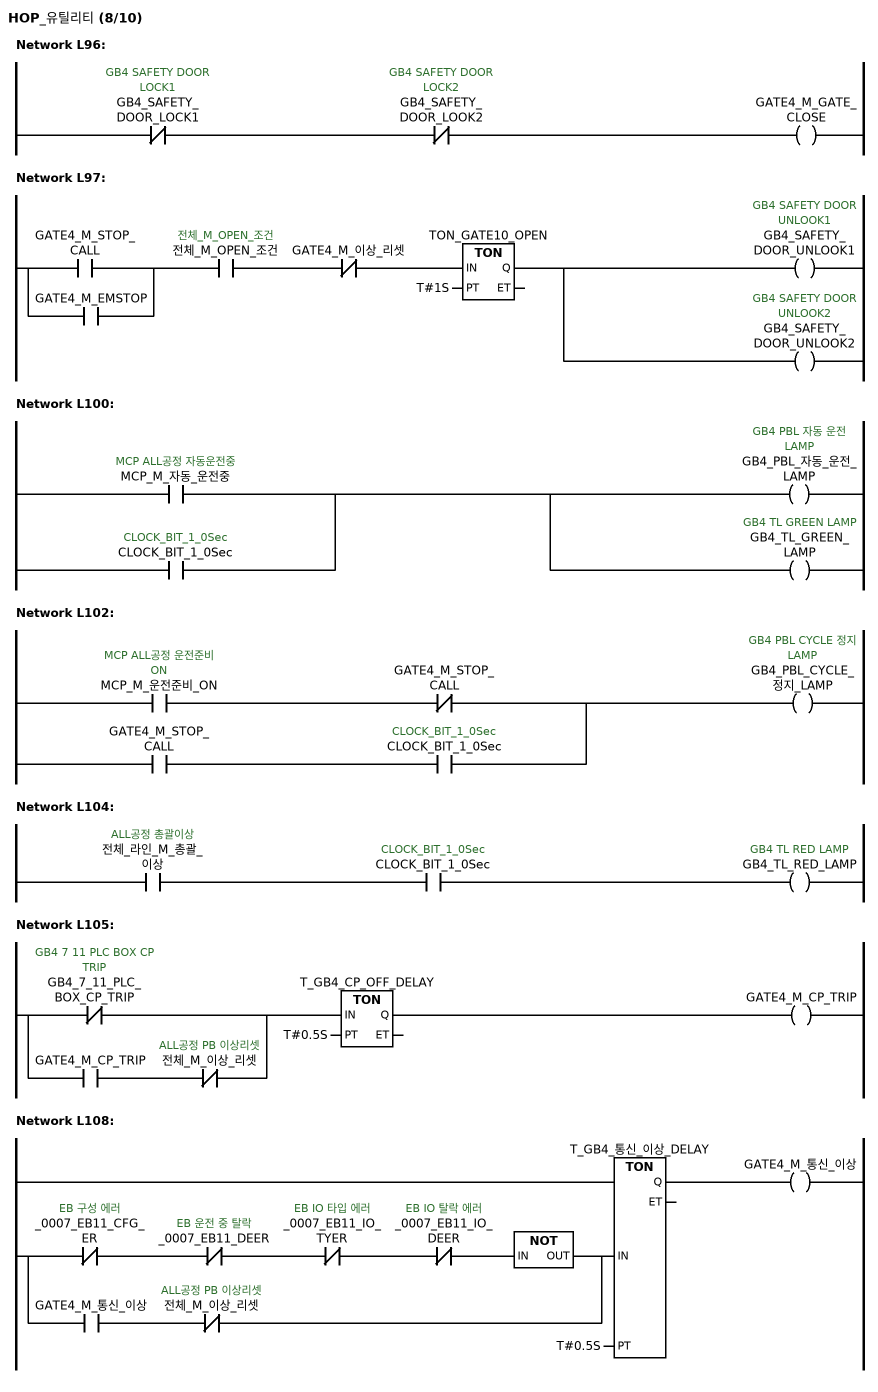
(* [picture p48: HOP_유틸리티 rungs L96-L108] *)
(* Rung L96 *)
GATE4_M_GATE_CLOSE := NOT GB4_SAFETY_DOOR_LOCK1 AND NOT GB4_SAFETY_DOOR_LOOK2;
(* Rung L97 *)
TON_GATE10_OPEN(IN := (GATE4_M_STOP_CALL OR GATE4_M_EMSTOP) AND 전체_M_OPEN_조건 AND NOT GATE4_M_이상_리셋, PT := T#1S);
GB4_SAFETY_DOOR_UNLOOK1 := TON_GATE10_OPEN.Q;
GB4_SAFETY_DOOR_UNLOOK2 := TON_GATE10_OPEN.Q;
(* Rung L100 *)
GB4_PBL_자동_운전_LAMP := MCP_M_자동_운전중 OR CLOCK_BIT_1_0Sec;
GB4_TL_GREEN_LAMP := MCP_M_자동_운전중 OR CLOCK_BIT_1_0Sec;
(* Rung L102 *)
GB4_PBL_CYCLE_정지_LAMP := (MCP_M_운전준비_ON AND NOT GATE4_M_STOP_CALL) OR (GATE4_M_STOP_CALL AND CLOCK_BIT_1_0Sec);
(* Rung L104 *)
GB4_TL_RED_LAMP := 전체_라인_M_총괄_이상 AND CLOCK_BIT_1_0Sec;
(* Rung L105 *)
T_GB4_CP_OFF_DELAY(IN := NOT GB4_7_11_PLC_BOX_CP_TRIP OR (GATE4_M_CP_TRIP AND NOT 전체_M_이상_리셋), PT := T#0.5S);
GATE4_M_CP_TRIP := T_GB4_CP_OFF_DELAY.Q;
(* Rung L108 *)
T_GB4_통신_이상_DELAY(IN := (NOT (NOT _0007_EB11_CFG_ER AND NOT _0007_EB11_DEER AND NOT _0007_EB11_IO_TYER AND NOT _0007_EB11_IO_DEER)) OR (GATE4_M_통신_이상 AND NOT 전체_M_이상_리셋), PT := T#0.5S);
GATE4_M_통신_이상 := T_GB4_통신_이상_DELAY.Q;

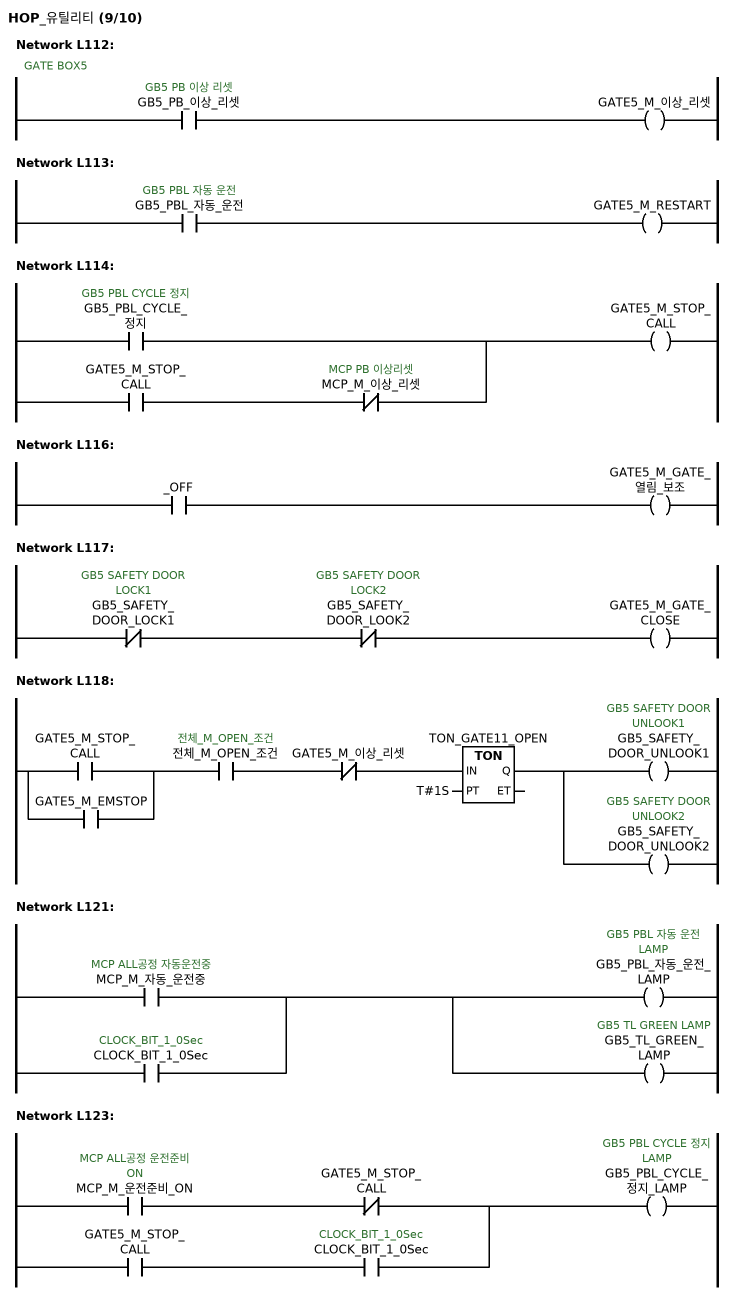
(* GATE BOX5 *)
(* Rung L112 *)
GATE5_M_이상_리셋 := GB5_PB_이상_리셋;
(* Rung L113 *)
GATE5_M_RESTART := GB5_PBL_자동_운전;
(* Rung L114 *)
GATE5_M_STOP_CALL := GB5_PBL_CYCLE_정지 OR (GATE5_M_STOP_CALL AND NOT MCP_M_이상_리셋);
(* Rung L116 *)
GATE5_M_GATE_열림_보조 := _OFF;
(* Rung L117 *)
GATE5_M_GATE_CLOSE := NOT GB5_SAFETY_DOOR_LOCK1 AND NOT GB5_SAFETY_DOOR_LOOK2;
(* Rung L118 *)
TON_GATE11_OPEN(IN := (GATE5_M_STOP_CALL OR GATE5_M_EMSTOP) AND 전체_M_OPEN_조건 AND NOT GATE5_M_이상_리셋, PT := T#1S);
GB5_SAFETY_DOOR_UNLOOK1 := TON_GATE11_OPEN.Q;
GB5_SAFETY_DOOR_UNLOOK2 := TON_GATE11_OPEN.Q;
(* Rung L121 *)
GB5_PBL_자동_운전_LAMP := MCP_M_자동_운전중 OR CLOCK_BIT_1_0Sec;
GB5_TL_GREEN_LAMP := MCP_M_자동_운전중 OR CLOCK_BIT_1_0Sec;
(* Rung L123 *)
GB5_PBL_CYCLE_정지_LAMP := (MCP_M_운전준비_ON AND NOT GATE5_M_STOP_CALL) OR (GATE5_M_STOP_CALL AND CLOCK_BIT_1_0Sec);

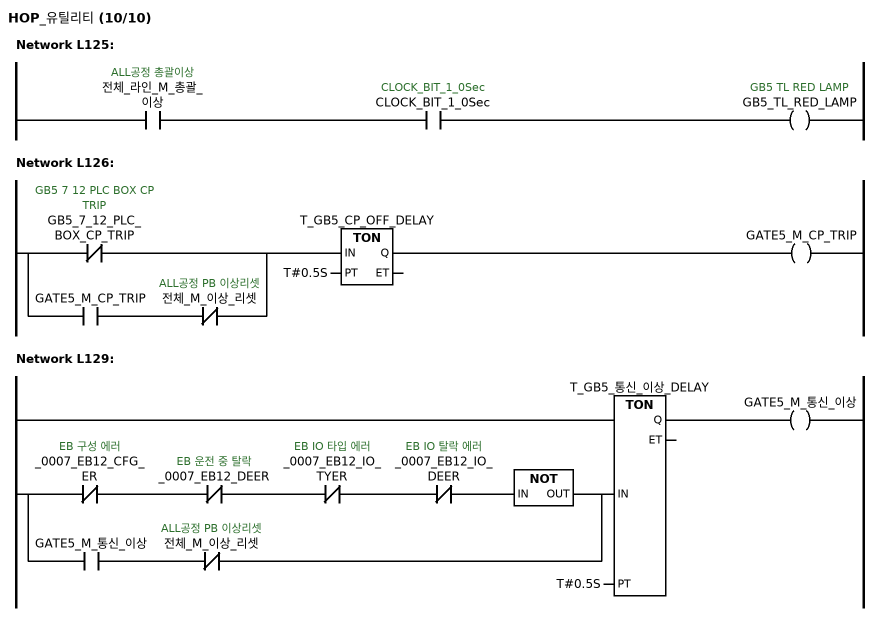
(* Rung L125 *)
GB5_TL_RED_LAMP := 전체_라인_M_총괄_이상 AND CLOCK_BIT_1_0Sec;
(* Rung L126 *)
T_GB5_CP_OFF_DELAY(IN := NOT GB5_7_12_PLC_BOX_CP_TRIP OR (GATE5_M_CP_TRIP AND NOT 전체_M_이상_리셋), PT := T#0.5S);
GATE5_M_CP_TRIP := T_GB5_CP_OFF_DELAY.Q;
(* Rung L129 *)
T_GB5_통신_이상_DELAY(IN := (NOT (NOT _0007_EB12_CFG_ER AND NOT _0007_EB12_DEER AND NOT _0007_EB12_IO_TYER AND NOT _0007_EB12_IO_DEER)) OR (GATE5_M_통신_이상 AND NOT 전체_M_이상_리셋), PT := T#0.5S);
GATE5_M_통신_이상 := T_GB5_통신_이상_DELAY.Q;
END_PROGRAM

PROGRAM 이상_총괄모음 (* task: 스캔 프로그램 *)
VAR_EXTERNAL RETAIN
    ALWAYS_OFF : BOOL; (* AT %MW3.0 *) (* 항시 OFF *)
    GATE1_M_CP_TRIP : BOOL; (* AT %MW400.15 *) (* GATEBOX1 CP OFF 이상 *)
    GATE1_M_EMSTOP : BOOL; (* AT %MW400.7 *) (* GATE1 비상정지 이상 *)
    GATE1_M_GATE_OPEN : BOOL; (* AT %MW400.13 *) (* GATEBOX1 이상 *)
    GATE1_M_통신_이상 : BOOL; (* AT %MW400.14 *) (* GATEBOX1 통신이상 *)
    GATE2_M_CP_TRIP : BOOL; (* AT %MW401.15 *) (* GATEBOX2 CP OFF 이상 *)
    GATE2_M_EMSTOP : BOOL; (* AT %MW401.7 *) (* GATE2 비상정지 이상 *)
    GATE2_M_GATE_OPEN : BOOL; (* AT %MW401.13 *) (* GATEBOX2 이상 *)
    GATE2_M_통신_이상 : BOOL; (* AT %MW401.14 *) (* GATEBOX2 통신이상 *)
    GATE3_M_CP_TRIP : BOOL; (* AT %MW402.15 *) (* GATEBOX3 CP OFF 이상 *)
    GATE3_M_EMSTOP : BOOL; (* AT %MW402.7 *) (* GATE3 비상정지 이상 *)
    GATE3_M_GATE_OPEN : BOOL; (* AT %MW402.13 *) (* GATEBOX3 이상 *)
    GATE3_M_통신_이상 : BOOL; (* AT %MW402.14 *) (* GATEBOX3 통신이상 *)
    GATE4_M_CP_TRIP : BOOL; (* AT %MW403.15 *)
    GATE4_M_EMSTOP : BOOL; (* AT %MW403.7 *)
    GATE4_M_GATE_OPEN : BOOL; (* AT %MW403.13 *)
    GATE4_M_통신_이상 : BOOL; (* AT %MW403.14 *)
    GATE5_M_CP_TRIP : BOOL; (* AT %MW404.15 *)
    GATE5_M_EMSTOP : BOOL; (* AT %MW404.7 *)
    GATE5_M_GATE_OPEN : BOOL; (* AT %MW404.13 *)
    GATE5_M_통신_이상 : BOOL; (* AT %MW404.14 *)
    HOP1_M_CP_OFF_이상 : BOOL; (* AT %MW360.15 *) (* HOP1 CP OFF 이상 *)
    HOP1_M_비상정지 : BOOL; (* AT %MW360.7 *) (* HOP1 비상정지 이상 *)
    HOP1_M_통신_이상 : BOOL; (* AT %MW360.14 *) (* HOP1 통신이상 *)
    INV1_M_CP_OFF_이상 : BOOL; (* AT %MW355.3 *) (* 인버터반1 CP OFF 이상 *)
    INV1_M_PS_DC_LOW : BOOL; (* AT %MW355.2 *) (* 인버터반1 PS저전압 이상 *)
    INV1_M_SPD_이상 : BOOL; (* AT %MW355.1 *) (* 인버터반1 SPD 이상 *)
    INV1_M_총괄_이상 : BOOL; (* AT %MW355.0 *) (* INV1_M_총괄_이상 *)
    INV1_M_통신_이상 : BOOL; (* AT %MW355.4 *) (* 인버터반1 통신이상 *)
    MCP_M_CP_OFF_이상 : BOOL; (* AT %MW351.0 *) (* MCP CP OFF 이상총괄 *)
    MCP_M_DISPLAY_CP_TRIP : BOOL; (* AT %MW351.6 *) (* MCP 출력전원 CP OFF 이상 *)
    MCP_M_HUB_CP_TRIP : BOOL; (* AT %MW351.1 *) (* MCP PS전원 CP OFF 이상 *)
    MCP_M_INPUT_CP_TRIP : BOOL; (* AT %MW351.3 *) (* MCP HUB전원  CP OFF 이상 *)
    MCP_M_OUTPUT_CP_TRIP : BOOL; (* AT %MW351.4 *) (* MCP 통신모듈 전원 CP OFF 이상 *)
    MCP_M_OUTPUT_MC_이상 : BOOL; (* AT %MW354.8 *) (* MCP 운전준비 MC 이상 *)
    MCP_M_PROFI_PWR_CP_TRIP : BOOL; (* AT %MW351.5 *) (* MCP 입력전원 CP OFF 이상 *)
    MCP_M_PS1_DC_LOW : BOOL; (* AT %MW353.1 *) (* MCP PS1 전원 이상 *)
    MCP_M_PS2_DC_LOW : BOOL; (* AT %MW353.2 *) (* MCP PS2 전원 이상 *)
    MCP_M_PS3_DC_LOW : BOOL; (* AT %MW353.3 *) (* MCP PS3 전원 이상 *)
    MCP_M_PS4_DC_LOW : BOOL; (* AT %MW353.4 *) (* MCP PS4 전원 이상 *)
    MCP_M_PS_DC_LOW : BOOL; (* AT %MW353.0 *) (* MCP PS 전원 이상총괄 *)
    MCP_M_SAG1_1_이상 : BOOL; (* AT %MW352.1 *) (* MCP SAG장치 이상 *)
    MCP_M_SAG1_2_이상 : BOOL; (* AT %MW352.2 *) (* MC SAG장치2 이상 *)
    MCP_M_SAG_이상 : BOOL; (* AT %MW352.0 *) (* MCP SAG장치 이상총괄 *)
    MCP_M_SPD_이상 : BOOL; (* AT %MW354.0 *) (* MCP 동력반 SPD 이상 *)
    MCP_M_비상정지 : BOOL; (* AT %MW350.7 *) (* MCP 비상정지 이상 *)
    MCP_M_이상_리셋 : BOOL; (* AT %MW350.4 *) (* MCP PB 이상리셋 *)
    MCP_M_통신_CP_TRIP : BOOL; (* AT %MW351.2 *) (* MCP   HMI전원  CP OFF 이상 *)
    MCP_M_통신_이상 : BOOL; (* AT %MW352.8 *) (* MCP 통신이상 *)
    S362_M_총괄_CP_이상 : BOOL; (* AT %MW1009.7 *) (* S362 CP OFF 이상 *)
    S362_M_총괄_CT_이상 : BOOL; (* AT %MW1010.4 *) (* S362   TACK TIME 이상 *)
    S362_M_총괄_INV_이상 : BOOL; (* AT %MW1009.9 *) (* S362 인버터 이상 *)
    S362_M_총괄_LS_이상 : BOOL; (* AT %MW1009.15 *) (* S362 LS 이상 *)
    S362_M_총괄_MATCH_이상 : BOOL; (* AT %MW1010.0 *) (* S362 매트SW 이상 *)
    S362_M_총괄_MC_이상 : BOOL; (* AT %MW1009.13 *) (* S362 MC 이상 *)
    S362_M_총괄_MOTOR_이상 : BOOL; (* AT %MW1010.3 *) (* S362 MOTOR 이상 *)
    S362_M_총괄_NFB_이상 : BOOL; (* AT %MW1009.11 *) (* S362 NFB 이상 *)
    S362_M_총괄_ROBOT_이상 : BOOL; (* AT %MW1010.1 *) (* S362 ROBOT 이상 *)
    S362_M_총괄_SAFETY_이상 : BOOL; (* AT %MW1009.2 *) (* S362 SAFETY 이상 *)
    S362_M_총괄_공기압_이상 : BOOL; (* AT %MW1009.3 *) (* S362 공기압 이상 *)
    S362_M_총괄_비상정지_이상 : BOOL; (* AT %MW1009.1 *) (* S362_M_총괄_비상정지_이상 *)
    S362_M_총괄_사양_이상 : BOOL; (* AT %MW1009.6 *) (* S362 사양 이상 *)
    S362_M_총괄_오버런_이상 : BOOL; (* AT %MW1009.12 *) (* S362 OVER RUN 이상 *)
    S362_M_총괄_용접타점수_이상 : BOOL; (* AT %MW1010.2 *) (* S362 용접타점수 이상 *)
    S362_M_총괄_제품감지_이상 : BOOL; (* AT %MW1009.4 *) (* S362 제품감지 이상 *)
    S362_M_총괄_차종_이상 : BOOL; (* AT %MW1009.5 *) (* S362 차종 이상 *)
    S362_M_총괄_통신_이상 : BOOL; (* AT %MW1009.14 *) (* S362 통신이상 *)
    S364_M_총괄_CP_이상 : BOOL; (* AT %MW2009.7 *) (* S364 CP OFF 이상 *)
    S364_M_총괄_CT_이상 : BOOL; (* AT %MW2010.4 *) (* S364   TACK TIME 이상 *)
    S364_M_총괄_LS_이상 : BOOL; (* AT %MW2009.15 *) (* S364 LS 이상 *)
    S364_M_총괄_MATCH_이상 : BOOL; (* AT %MW2010.0 *) (* S364 매트SW 이상 *)
    S364_M_총괄_ROBOT_이상 : BOOL; (* AT %MW2010.1 *) (* S364 ROBOT 이상 *)
    S364_M_총괄_SAFETY_이상 : BOOL; (* AT %MW2009.2 *) (* S364 SAFETY 이상 *)
    S364_M_총괄_공기압_이상 : BOOL; (* AT %MW2009.3 *) (* S364 공기압 이상 *)
    S364_M_총괄_비상정지_이상 : BOOL; (* AT %MW2009.1 *) (* S364_M_총괄_비상정지_이상 *)
    S364_M_총괄_사양_이상 : BOOL; (* AT %MW2009.6 *) (* S364 사양 이상 *)
    S364_M_총괄_용접타점수_이상 : BOOL; (* AT %MW2010.2 *) (* S364 용접타점수 이상 *)
    S364_M_총괄_제품감지_이상 : BOOL; (* AT %MW2009.4 *) (* S364 제품감지 이상 *)
    S364_M_총괄_차종_이상 : BOOL; (* AT %MW2009.5 *) (* S364 차종 이상 *)
    S364_M_총괄_통신_이상 : BOOL; (* AT %MW2009.14 *) (* S364 통신이상 *)
    S365_M_총괄_CP_이상 : BOOL; (* AT %MW2509.7 *) (* S365 CP OFF 이상 *)
    S365_M_총괄_CT_이상 : BOOL; (* AT %MW2510.4 *) (* S365   TACK TIME 이상 *)
    S365_M_총괄_LS_이상 : BOOL; (* AT %MW2509.15 *) (* S365 LS 이상 *)
    S365_M_총괄_MATCH_이상 : BOOL; (* AT %MW2510.0 *) (* S365 매트SW 이상 *)
    S365_M_총괄_ROBOT_이상 : BOOL; (* AT %MW2510.1 *) (* S365 ROBOT 이상 *)
    S365_M_총괄_SAFETY_이상 : BOOL; (* AT %MW2509.2 *) (* S365 SAFETY 이상 *)
    S365_M_총괄_공기압_이상 : BOOL; (* AT %MW2509.3 *) (* S365 공기압 이상 *)
    S365_M_총괄_비상정지_이상 : BOOL; (* AT %MW2509.1 *) (* S365_M_총괄_비상정지_이상 *)
    S365_M_총괄_사양_이상 : BOOL; (* AT %MW2509.6 *) (* S365 사양 이상 *)
    S365_M_총괄_용접타점수_이상 : BOOL; (* AT %MW2510.2 *) (* S365 용접타점수 이상 *)
    S365_M_총괄_제품감지_이상 : BOOL; (* AT %MW2509.4 *) (* S365 제품감지 이상 *)
    S365_M_총괄_차종_이상 : BOOL; (* AT %MW2509.5 *) (* S365 차종 이상 *)
    S365_M_총괄_통신_이상 : BOOL; (* AT %MW2509.14 *) (* S365 통신이상 *)
    S366_M_총괄_CP_이상 : BOOL; (* AT %MW3009.7 *) (* S366 CP OFF 이상 *)
    S366_M_총괄_CT_이상 : BOOL; (* AT %MW3010.4 *) (* S366   TACK TIME 이상 *)
    S366_M_총괄_INV_이상 : BOOL; (* AT %MW3009.9 *) (* S366 인버터 이상 *)
    S366_M_총괄_LS_이상 : BOOL; (* AT %MW3009.15 *) (* S366 LS 이상 *)
    S366_M_총괄_MATCH_이상 : BOOL; (* AT %MW3010.0 *) (* S366 매트SW 이상 *)
    S366_M_총괄_MC_이상 : BOOL; (* AT %MW3009.13 *) (* S366 MC 이상 *)
    S366_M_총괄_MOTOR_이상 : BOOL; (* AT %MW3010.3 *) (* S366 MOTOR 이상 *)
    S366_M_총괄_NFB_이상 : BOOL; (* AT %MW3009.11 *) (* S366 NFB 이상 *)
    S366_M_총괄_ROBOT_이상 : BOOL; (* AT %MW3010.1 *) (* S366 ROBOT 이상 *)
    S366_M_총괄_SAFETY_이상 : BOOL; (* AT %MW3009.2 *) (* S366_M_총괄_SAFETY_이상 *)
    S366_M_총괄_공기압_이상 : BOOL; (* AT %MW3009.3 *) (* S366 공기압 이상 *)
    S366_M_총괄_비상정지_이상 : BOOL; (* AT %MW3009.1 *) (* S366_M_총괄_비상정지_이상 *)
    S366_M_총괄_사양_이상 : BOOL; (* AT %MW3009.6 *) (* S366 사양 이상 *)
    S366_M_총괄_오버런_이상 : BOOL; (* AT %MW3009.12 *) (* S366 OVER RUN 이상 *)
    S366_M_총괄_용접타점수_이상 : BOOL; (* AT %MW3010.2 *) (* S366 용접타점수 이상 *)
    S366_M_총괄_제품감지_이상 : BOOL; (* AT %MW3009.4 *) (* S366 제품감지 이상 *)
    S366_M_총괄_차종_이상 : BOOL; (* AT %MW3009.5 *) (* S366 차종 이상 *)
    S366_M_총괄_통신_이상 : BOOL; (* AT %MW3009.14 *) (* S366 통신이상 *)
    S367_M_총괄_CP_이상 : BOOL; (* AT %MW3509.7 *) (* S367 CP OFF 이상 *)
    S367_M_총괄_CT_이상 : BOOL; (* AT %MW3510.4 *) (* S367   TACK TIME 이상 *)
    S367_M_총괄_LS_이상 : BOOL; (* AT %MW3509.15 *) (* S367 LS 이상 *)
    S367_M_총괄_MATCH_이상 : BOOL; (* AT %MW3510.0 *) (* S367 매트SW 이상 *)
    S367_M_총괄_ROBOT_이상 : BOOL; (* AT %MW3510.1 *) (* S367 ROBOT 이상 *)
    S367_M_총괄_SAFETY_이상 : BOOL; (* AT %MW3509.2 *) (* S367_M_총괄_SAFETY_이상 *)
    S367_M_총괄_공기압_이상 : BOOL; (* AT %MW3509.3 *) (* S367 공기압 이상 *)
    S367_M_총괄_비상정지_이상 : BOOL; (* AT %MW3509.1 *) (* S367_M_총괄_비상정지_이상 *)
    S367_M_총괄_사양_이상 : BOOL; (* AT %MW3509.6 *) (* S367 사양 이상 *)
    S367_M_총괄_용접타점수_이상 : BOOL; (* AT %MW3510.2 *) (* S367 용접타점수 이상 *)
    S367_M_총괄_제품감지_이상 : BOOL; (* AT %MW3509.4 *) (* S367 제품감지 이상 *)
    S367_M_총괄_차종_이상 : BOOL; (* AT %MW3509.5 *) (* S367 차종 이상 *)
    S367_M_총괄_통신_이상 : BOOL; (* AT %MW3509.14 *) (* S367 통신이상 *)
    S368_M_총괄_CP_이상 : BOOL; (* AT %MW4009.7 *) (* S368 CP OFF 이상 *)
    S368_M_총괄_CT_이상 : BOOL; (* AT %MW4010.4 *) (* S368   TACK TIME 이상 *)
    S368_M_총괄_LS_이상 : BOOL; (* AT %MW4009.15 *) (* S368 LS 이상 *)
    S368_M_총괄_MATCH_이상 : BOOL; (* AT %MW4010.0 *) (* S368 매트SW 이상 *)
    S368_M_총괄_ROBOT_이상 : BOOL; (* AT %MW4010.1 *) (* S368 ROBOT 이상 *)
    S368_M_총괄_SAFETY_이상 : BOOL; (* AT %MW4009.2 *) (* S368_M_총괄_SAFETY_이상 *)
    S368_M_총괄_공기압_이상 : BOOL; (* AT %MW4009.3 *) (* S368 공기압 이상 *)
    S368_M_총괄_비상정지_이상 : BOOL; (* AT %MW4009.1 *) (* S368_M_총괄_비상정지_이상 *)
    S368_M_총괄_사양_이상 : BOOL; (* AT %MW4009.6 *) (* S368 사양 이상 *)
    S368_M_총괄_용접타점수_이상 : BOOL; (* AT %MW4010.2 *) (* S368 용접타점수 이상 *)
    S368_M_총괄_제품감지_이상 : BOOL; (* AT %MW4009.4 *) (* S368 제품감지 이상 *)
    S368_M_총괄_차종_이상 : BOOL; (* AT %MW4009.5 *) (* S368 차종 이상 *)
    S368_M_총괄_통신_이상 : BOOL; (* AT %MW4009.14 *) (* S368 통신이상 *)
    S369_1_M_총괄_CP_이상 : BOOL; (* AT %MW4509.7 *) (* S369-1 CP OFF 이상 *)
    S369_1_M_총괄_CT_이상 : BOOL; (* AT %MW4510.4 *) (* S369-1 TACK TIME 이상 *)
    S369_1_M_총괄_LS_이상 : BOOL; (* AT %MW4509.15 *) (* S369-1 LS 이상 *)
    S369_1_M_총괄_MATCH_이상 : BOOL; (* AT %MW4510.0 *) (* S369-1 매트SW 이상 *)
    S369_1_M_총괄_ROBOT_이상 : BOOL; (* AT %MW4510.1 *) (* S369-1 ROBOT 이상 *)
    S369_1_M_총괄_SAFETY_이상 : BOOL; (* AT %MW4509.2 *) (* S369_1_M_총괄_SAFETY_이상 *)
    S369_1_M_총괄_공기압_이상 : BOOL; (* AT %MW4509.3 *) (* S36-1 공기압 이상 *)
    S369_1_M_총괄_사양_이상 : BOOL; (* AT %MW4509.6 *) (* S369-1 사양 이상 *)
    S369_1_M_총괄_용접타점수_이상 : BOOL; (* AT %MW4510.2 *) (* S369-1 용접타점수 이상 *)
    S369_1_M_총괄_제품감지_이상 : BOOL; (* AT %MW4509.4 *) (* S369-1 제품감지 이상 *)
    S369_1_M_총괄_차종_이상 : BOOL; (* AT %MW4509.5 *) (* S369-1 차종 이상 *)
    S369_1_M_총괄_통신_이상 : BOOL; (* AT %MW4509.14 *) (* S369-1 통신이상 *)
    S369_M_총괄_CP_이상 : BOOL; (* AT %MW5009.7 *) (* S369 CP OFF 이상 *)
    S369_M_총괄_CT_이상 : BOOL; (* AT %MW5010.4 *) (* S369   TACK TIME 이상 *)
    S369_M_총괄_LS_이상 : BOOL; (* AT %MW5009.15 *) (* S369 LS 이상 *)
    S369_M_총괄_MATCH_이상 : BOOL; (* AT %MW5010.0 *) (* S369 매트SW 이상 *)
    S369_M_총괄_MOTOR_이상 : BOOL; (* AT %MW5010.3 *) (* S369 MOTOR 이상 *)
    S369_M_총괄_NFB_이상 : BOOL; (* AT %MW5009.11 *) (* S369 NFB 이상 *)
    S369_M_총괄_ROBOT_이상 : BOOL; (* AT %MW5010.1 *) (* S369 ROBOT 이상 *)
    S369_M_총괄_SAFETY_이상 : BOOL; (* AT %MW5009.2 *) (* S369_M_총괄_SAFETY_이상 *)
    S369_M_총괄_SRV_이상 : BOOL; (* AT %MW5009.10 *) (* S369 SERVO 이상 *)
    S369_M_총괄_공기압_이상 : BOOL; (* AT %MW5009.3 *) (* S369 공기압 이상 *)
    S369_M_총괄_비상정지_이상 : BOOL; (* AT %MW5009.1 *) (* S369_M_총괄_비상정지_이상 *)
    S369_M_총괄_사양_이상 : BOOL; (* AT %MW5009.6 *) (* S369 사양 이상 *)
    S369_M_총괄_오버런_이상 : BOOL; (* AT %MW5009.12 *) (* S369 OVER RUN 이상 *)
    S369_M_총괄_용접타점수_이상 : BOOL; (* AT %MW5010.2 *) (* S369 용접타점수 이상 *)
    S369_M_총괄_제품감지_이상 : BOOL; (* AT %MW5009.4 *) (* S369 제품감지 이상 *)
    S369_M_총괄_차종_이상 : BOOL; (* AT %MW5009.5 *) (* S369 차종 이상 *)
    S369_M_총괄_통신_이상 : BOOL; (* AT %MW5009.14 *) (* S369 통신이상 *)
    SRV1_M_CP_OFF_이상 : BOOL; (* AT %MW356.3 *) (* 서보반1 CP OFF 이상 *)
    SRV1_M_PS_DC_LOW : BOOL; (* AT %MW356.2 *) (* 서보반1 PS저전압 이상 *)
    SRV1_M_SPD_이상 : BOOL; (* AT %MW356.1 *) (* 서보반1 SPD 이상 *)
    SRV1_M_총괄_이상 : BOOL; (* AT %MW356.0 *) (* SRV1_M_총괄_이상 *)
    SRV1_M_통신_이상 : BOOL; (* AT %MW356.4 *) (* SERVO반1 통신이상 *)
    전체_라인_M_총괄_CP_OFF : BOOL; (* AT %MW300.7 *) (* ALL공정 CP OFF 이상총괄 *)
    전체_라인_M_총괄_CT_이상 : BOOL; (* AT %MW301.4 *) (* ALL공정 TACK TIME 이상총괄 *)
    전체_라인_M_총괄_EOCR_이상 : BOOL; (* AT %MW300.8 *) (* ALL공정 EOCR 이상총괄 *)
    전체_라인_M_총괄_GATE_OPEN_이상 : BOOL; (* AT %MW301.5 *) (* ALL공정 GATEBOX 이상총괄 *)
    전체_라인_M_총괄_INV_이상 : BOOL; (* AT %MW300.9 *) (* ALL공정 인버터 이상총괄 *)
    전체_라인_M_총괄_LS_이상 : BOOL; (* AT %MW300.15 *) (* ALL공정 LS 이상총괄 *)
    전체_라인_M_총괄_MATCH_이상 : BOOL; (* AT %MW301.0 *) (* ALL공정 매트SW 이상총괄 *)
    전체_라인_M_총괄_MC_이상 : BOOL; (* AT %MW300.13 *) (* ALL공정 MC 이상총괄 *)
    전체_라인_M_총괄_MOTOR_이상 : BOOL; (* AT %MW301.3 *) (* ALL공정 MOTOR 이상총괄 *)
    전체_라인_M_총괄_NFB_이상 : BOOL; (* AT %MW300.11 *) (* ALL공정 NFB 이상총괄 *)
    전체_라인_M_총괄_PS_DC_LOW : BOOL; (* AT %MW301.7 *) (* ALL공정 PS저전압 이상총괄 *)
    전체_라인_M_총괄_ROBOT_이상 : BOOL; (* AT %MW301.1 *) (* ALL공정 ROBOT 총괄이상 *)
    전체_라인_M_총괄_SAFETY_이상 : BOOL; (* AT %MW300.2 *) (* ALL공정 SAFETY  이상총괄 *)
    전체_라인_M_총괄_SAG_이상 : BOOL; (* AT %MW301.6 *) (* ALL공정 SAG 이상총괄 *)
    전체_라인_M_총괄_SPD_이상 : BOOL; (* AT %MW301.8 *) (* ALL공정 SPD 이상총괄 *)
    전체_라인_M_총괄_SRV_이상 : BOOL; (* AT %MW300.10 *) (* ALL공정 SERVO 이상총괄 *)
    전체_라인_M_총괄_공기압_이상 : BOOL; (* AT %MW300.3 *) (* ALL공정 공기압 이상총괄 *)
    전체_라인_M_총괄_비상정지_이상 : BOOL; (* AT %MW300.1 *) (* ALL공정 비상정지 이상총괄 *)
    전체_라인_M_총괄_사양_이상 : BOOL; (* AT %MW300.6 *) (* ALL공정 사양 이상총괄 *)
    전체_라인_M_총괄_오버런_이상 : BOOL; (* AT %MW300.12 *) (* ALL공정 OVER RUN 이상총괄 *)
    전체_라인_M_총괄_용접타점수_이상 : BOOL; (* AT %MW301.2 *) (* ALL공정 용접타점수 이상총괄 *)
    전체_라인_M_총괄_이상 : BOOL; (* AT %MW300.0 *) (* ALL공정 총괄이상 *)
    전체_라인_M_총괄_제품감지_이상 : BOOL; (* AT %MW300.4 *) (* ALL공정 제품감지 이상총괄 *)
    전체_라인_M_총괄_차종_이상 : BOOL; (* AT %MW300.5 *) (* ALL공정 차종 이상총괄 *)
    전체_라인_M_총괄_통신_이상 : BOOL; (* AT %MW300.14 *) (* ALL공정 통신 이상총괄 *)
END_VAR
VAR_EXTERNAL
    EGIS_ON : BOOL; (* 항시ON (임시용) *)
    MCP_DISPLAY_CP_TRIP : BOOL; (* AT %MW87632.5 *) (* MCP 출력전원 CP TRIP *)
    MCP_HUB_CP_TRIP : BOOL; (* AT %MW87632.0 *) (* MCP PS1전원  CP TRIP *)
    MCP_INPUT_PWR_CP_TRIP : BOOL; (* AT %MW87632.2 *) (* MCP HUB전원  CP TRIP *)
    MCP_OUTPUT_PWR_CP1_TRIP : BOOL; (* AT %MW87632.3 *) (* MCP 통신모듈 전원 CP TRIP *)
    MCP_OUTPUT_PWR_CP2_TRIP : BOOL; (* AT %MW87632.4 *) (* MCP 입력전원 CP TRIP *)
    MCP_PS1_DC_OK : BOOL; (* AT %MW87631.12 *) (* MCP PS1 전원 정상 *)
    MCP_PS2_DC_OK : BOOL; (* AT %MW87631.13 *) (* MCP PS2 전원 정상 *)
    MCP_PS3_DC_OK : BOOL; (* AT %MW87631.14 *) (* MCP PS3 전원 정상 *)
    MCP_PS4_DC_OK : BOOL; (* AT %MW87631.15 *) (* MCP PS4 전원 정상 *)
    MCP_SAFTY_MC_ON : BOOL; (* AT %MW87632.9 *) (* MCP 운전준비 MC 보조접점 *)
    MCP_운전준비_MC_ON : BOOL; (* AT %MW97636.0 *) (* MCP 운전준비 MC ON *)
    MCP_통신_CP_TRIP : BOOL; (* AT %MW87632.1 *) (* MCP HMI전원  CP TRIP *)
    PWR_SAG1_DSUB1_NOMAL1 : BOOL; (* AT %MW87631.10 *) (* MCP SAG장치 정상 *)
    PWR_SAG1_DSUB8_NOMAL2 : BOOL; (* AT %MW87631.11 *) (* MCP SAG장치 이상 *)
    PWR_SPD1_NOMAL : BOOL; (* AT %MW87631.8 *) (* MCP 동력반 SPD 정상 *)
    S362_6_INV_BRAKE_CP_OFF : BOOL; (* AT %MW85013.13 *) (* S362_6_INV_BRAKE_CP_OFF *)
    S362_6_INV_DC_CP_TRIP : BOOL; (* AT %MW85013.12 *) (* S362_6_INV_DC_CP_TRIP *)
    S362_6_INV_PS1_DC_OK : BOOL; (* AT %MW85013.14 *) (* S362_6_INV_PS1_DC_OK *)
    S362_6_INV_SPD_NOMAL : BOOL; (* AT %MW85013.15 *) (* S362_6_INV_SPD_NOMAL *)
    S362_6_INV_제어_CP_OFF : BOOL; (* AT %MW85013.11 *) (* S362_6_INV_제어_CP_OFF *)
    SERVO_PNL_SPD_NOMAL : BOOL; (* AT %MW85023.14 *) (* SERVO_PNL_SPD_NOMAL *)
    SERVO_PS1_1_DC_OK : BOOL; (* AT %MW85023.12 *) (* SERVO_PS1_1_DC_OK *)
    SERVO_PS1_2_DC_OK : BOOL; (* AT %MW85023.13 *) (* SERVO_PS1_2_DC_OK *)
    SERVO_PS_CP_TRIP : BOOL; (* AT %MW85023.15 *) (* SERVO_PS_CP_TRIP *)
    _MW87632_06 : BOOL; (* AT %MW87632.6 *) (* MCP 출력전원 CP TRIP *)
    _MW87632_07 : BOOL; (* AT %MW87632.7 *) (* MCP PC랙전원 CP TRIP *)
    _MW87632_08 : BOOL; (* AT %MW87632.8 *) (* MCP 현황판 CP TRIP *)
END_VAR
VAR
    INST1 : TON;
    INST10 : TON;
    INST11 : TON;
    INST12 : TON;
    INST13 : TON;
    INST14 : TON;
    INST15 : TON;
    INST16 : TON;
    INST17 : TON;
    INST18 : TON;
    INST19 : TON;
    INST2 : TON;
    INST20 : TON;
    INST21 : TON;
    INST22 : TON;
    INST23 : TON;
    INST24 : TON;
    INST25 : TON;
    INST26 : TON;
    INST27 : TON;
    INST3 : TON;
    INST4 : TON;
    INST5 : TON;
    INST6 : TON;
    INST7 : TON;
    INST8 : TON;
    INST9 : TON;
END_VAR

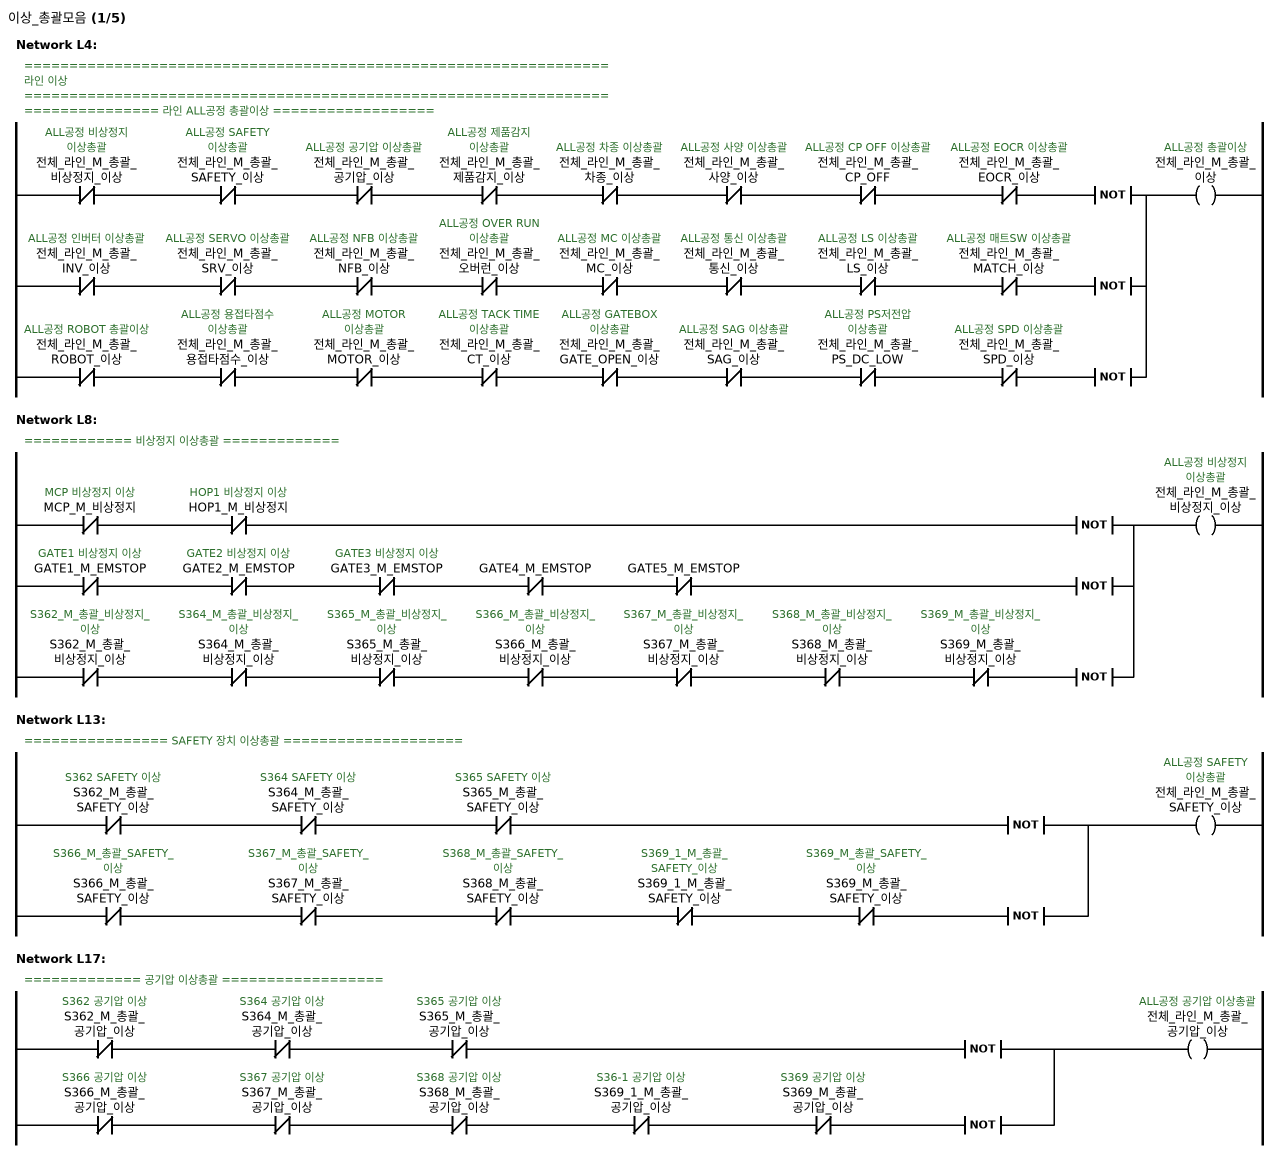
(* ================================================================= *)
(* 라인 이상 *)
(* ================================================================= *)
(* =============== 라인 ALL공정 총괄이상 ================== *)
(* Rung L4 *)
전체_라인_M_총괄_이상 := NOT (NOT 전체_라인_M_총괄_비상정지_이상 AND NOT 전체_라인_M_총괄_SAFETY_이상 AND NOT 전체_라인_M_총괄_공기압_이상 AND NOT 전체_라인_M_총괄_제품감지_이상 AND NOT 전체_라인_M_총괄_차종_이상 AND NOT 전체_라인_M_총괄_사양_이상 AND NOT 전체_라인_M_총괄_CP_OFF AND NOT 전체_라인_M_총괄_EOCR_이상) OR NOT (NOT 전체_라인_M_총괄_INV_이상 AND NOT 전체_라인_M_총괄_SRV_이상 AND NOT 전체_라인_M_총괄_NFB_이상 AND NOT 전체_라인_M_총괄_오버런_이상 AND NOT 전체_라인_M_총괄_MC_이상 AND NOT 전체_라인_M_총괄_통신_이상 AND NOT 전체_라인_M_총괄_LS_이상 AND NOT 전체_라인_M_총괄_MATCH_이상) OR NOT (NOT 전체_라인_M_총괄_ROBOT_이상 AND NOT 전체_라인_M_총괄_용접타점수_이상 AND NOT 전체_라인_M_총괄_MOTOR_이상 AND NOT 전체_라인_M_총괄_CT_이상 AND NOT 전체_라인_M_총괄_GATE_OPEN_이상 AND NOT 전체_라인_M_총괄_SAG_이상 AND NOT 전체_라인_M_총괄_PS_DC_LOW AND NOT 전체_라인_M_총괄_SPD_이상);
(* ============ 비상정지 이상총괄 ============= *)
(* Rung L8 *)
전체_라인_M_총괄_비상정지_이상 := NOT (NOT MCP_M_비상정지 AND NOT HOP1_M_비상정지) OR NOT (NOT GATE1_M_EMSTOP AND NOT GATE2_M_EMSTOP AND NOT GATE3_M_EMSTOP AND NOT GATE4_M_EMSTOP AND NOT GATE5_M_EMSTOP) OR NOT (NOT S362_M_총괄_비상정지_이상 AND NOT S364_M_총괄_비상정지_이상 AND NOT S365_M_총괄_비상정지_이상 AND NOT S366_M_총괄_비상정지_이상 AND NOT S367_M_총괄_비상정지_이상 AND NOT S368_M_총괄_비상정지_이상 AND NOT S369_M_총괄_비상정지_이상);
(* ================ SAFETY 장치 이상총괄 ==================== *)
(* Rung L13 *)
전체_라인_M_총괄_SAFETY_이상 := NOT (NOT S362_M_총괄_SAFETY_이상 AND NOT S364_M_총괄_SAFETY_이상 AND NOT S365_M_총괄_SAFETY_이상) OR NOT (NOT S366_M_총괄_SAFETY_이상 AND NOT S367_M_총괄_SAFETY_이상 AND NOT S368_M_총괄_SAFETY_이상 AND NOT S369_1_M_총괄_SAFETY_이상 AND NOT S369_M_총괄_SAFETY_이상);
(* ============= 공기압 이상총괄 ================== *)
(* Rung L17 *)
전체_라인_M_총괄_공기압_이상 := NOT (NOT S362_M_총괄_공기압_이상 AND NOT S364_M_총괄_공기압_이상 AND NOT S365_M_총괄_공기압_이상) OR NOT (NOT S366_M_총괄_공기압_이상 AND NOT S367_M_총괄_공기압_이상 AND NOT S368_M_총괄_공기압_이상 AND NOT S369_1_M_총괄_공기압_이상 AND NOT S369_M_총괄_공기압_이상);

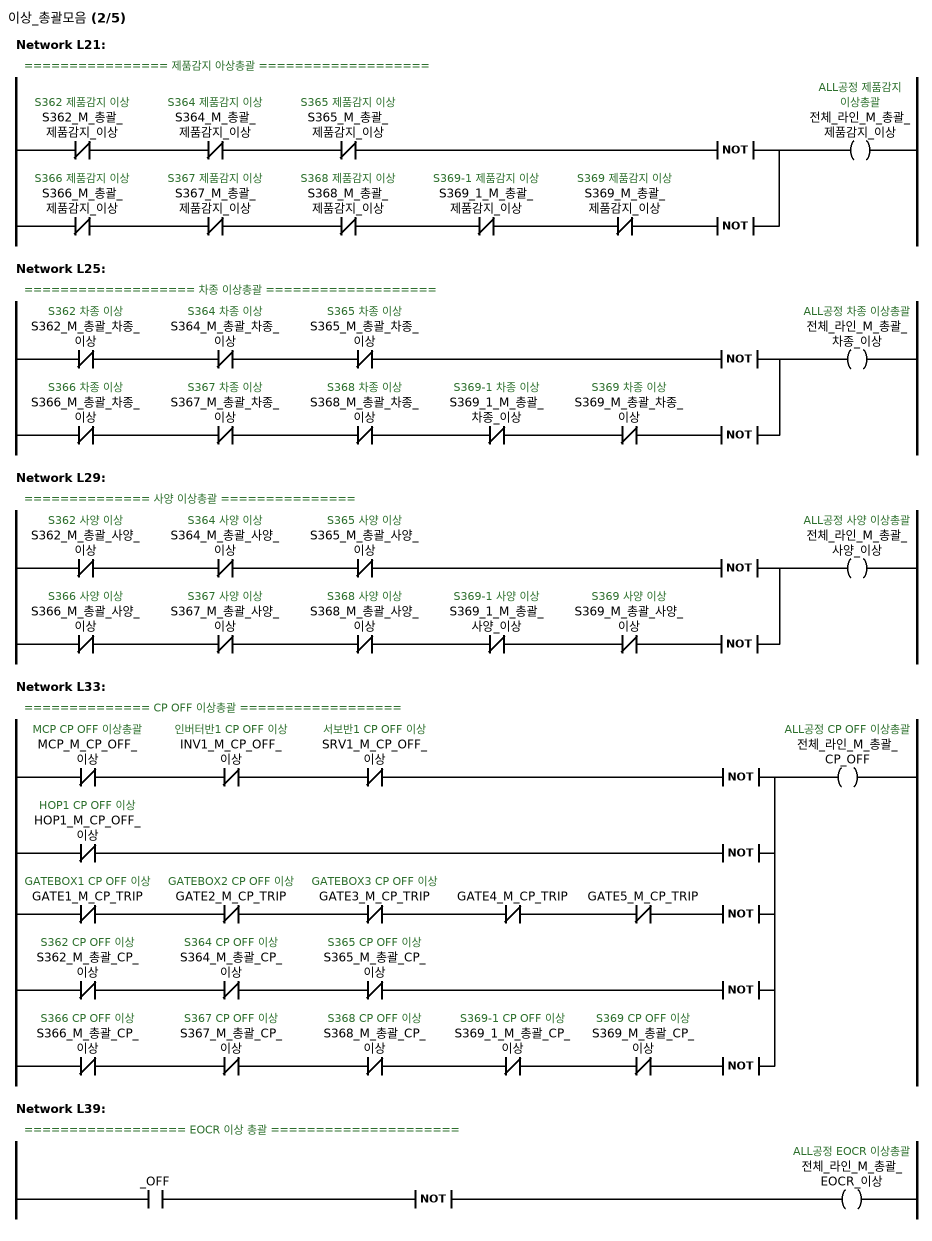
(* ================ 제품감지 아상총괄 =================== *)
(* Rung L21 *)
전체_라인_M_총괄_제품감지_이상 := NOT (NOT S362_M_총괄_제품감지_이상 AND NOT S364_M_총괄_제품감지_이상 AND NOT S365_M_총괄_제품감지_이상) OR NOT (NOT S366_M_총괄_제품감지_이상 AND NOT S367_M_총괄_제품감지_이상 AND NOT S368_M_총괄_제품감지_이상 AND NOT S369_1_M_총괄_제품감지_이상 AND NOT S369_M_총괄_제품감지_이상);
(* =================== 차종 이상총괄 =================== *)
(* Rung L25 *)
전체_라인_M_총괄_차종_이상 := NOT (NOT S362_M_총괄_차종_이상 AND NOT S364_M_총괄_차종_이상 AND NOT S365_M_총괄_차종_이상) OR NOT (NOT S366_M_총괄_차종_이상 AND NOT S367_M_총괄_차종_이상 AND NOT S368_M_총괄_차종_이상 AND NOT S369_1_M_총괄_차종_이상 AND NOT S369_M_총괄_차종_이상);
(* ============== 사양 이상총괄 =============== *)
(* Rung L29 *)
전체_라인_M_총괄_사양_이상 := NOT (NOT S362_M_총괄_사양_이상 AND NOT S364_M_총괄_사양_이상 AND NOT S365_M_총괄_사양_이상) OR NOT (NOT S366_M_총괄_사양_이상 AND NOT S367_M_총괄_사양_이상 AND NOT S368_M_총괄_사양_이상 AND NOT S369_1_M_총괄_사양_이상 AND NOT S369_M_총괄_사양_이상);
(* ============== CP OFF 이상총괄 ================== *)
(* Rung L33 *)
전체_라인_M_총괄_CP_OFF := NOT (NOT MCP_M_CP_OFF_이상 AND NOT INV1_M_CP_OFF_이상 AND NOT SRV1_M_CP_OFF_이상) OR HOP1_M_CP_OFF_이상 OR NOT (NOT GATE1_M_CP_TRIP AND NOT GATE2_M_CP_TRIP AND NOT GATE3_M_CP_TRIP AND NOT GATE4_M_CP_TRIP AND NOT GATE5_M_CP_TRIP) OR NOT (NOT S362_M_총괄_CP_이상 AND NOT S364_M_총괄_CP_이상 AND NOT S365_M_총괄_CP_이상) OR NOT (NOT S366_M_총괄_CP_이상 AND NOT S367_M_총괄_CP_이상 AND NOT S368_M_총괄_CP_이상 AND NOT S369_1_M_총괄_CP_이상 AND NOT S369_M_총괄_CP_이상);
(* ================== EOCR 이상 총괄 ===================== *)
(* Rung L39 *)
전체_라인_M_총괄_EOCR_이상 := NOT _OFF;

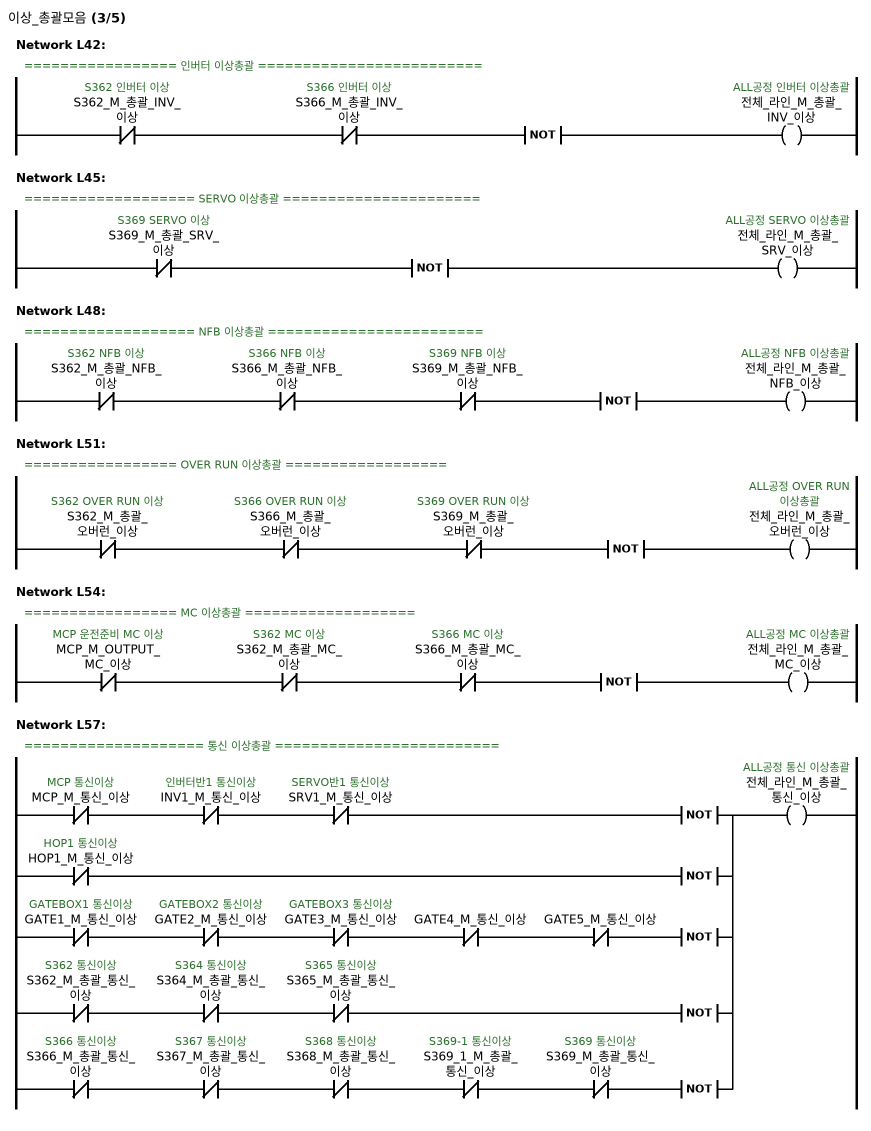
(* ================= 인버터 이상총괄 ========================= *)
(* Rung L42 *)
전체_라인_M_총괄_INV_이상 := NOT (NOT S362_M_총괄_INV_이상 AND NOT S366_M_총괄_INV_이상);
(* =================== SERVO 이상총괄 ====================== *)
(* Rung L45 *)
전체_라인_M_총괄_SRV_이상 := S369_M_총괄_SRV_이상;
(* =================== NFB 이상총괄 ======================== *)
(* Rung L48 *)
전체_라인_M_총괄_NFB_이상 := NOT (NOT S362_M_총괄_NFB_이상 AND NOT S366_M_총괄_NFB_이상 AND NOT S369_M_총괄_NFB_이상);
(* ================= OVER RUN 이상총괄 ================== *)
(* Rung L51 *)
전체_라인_M_총괄_오버런_이상 := NOT (NOT S362_M_총괄_오버런_이상 AND NOT S366_M_총괄_오버런_이상 AND NOT S369_M_총괄_오버런_이상);
(* ================= MC 이상총괄 =================== *)
(* Rung L54 *)
전체_라인_M_총괄_MC_이상 := NOT (NOT MCP_M_OUTPUT_MC_이상 AND NOT S362_M_총괄_MC_이상 AND NOT S366_M_총괄_MC_이상);
(* ==================== 통신 이상총괄 ========================= *)
(* Rung L57 *)
전체_라인_M_총괄_통신_이상 := NOT (NOT MCP_M_통신_이상 AND NOT INV1_M_통신_이상 AND NOT SRV1_M_통신_이상) OR HOP1_M_통신_이상 OR NOT (NOT GATE1_M_통신_이상 AND NOT GATE2_M_통신_이상 AND NOT GATE3_M_통신_이상 AND NOT GATE4_M_통신_이상 AND NOT GATE5_M_통신_이상) OR NOT (NOT S362_M_총괄_통신_이상 AND NOT S364_M_총괄_통신_이상 AND NOT S365_M_총괄_통신_이상) OR NOT (NOT S366_M_총괄_통신_이상 AND NOT S367_M_총괄_통신_이상 AND NOT S368_M_총괄_통신_이상 AND NOT S369_1_M_총괄_통신_이상 AND NOT S369_M_총괄_통신_이상);

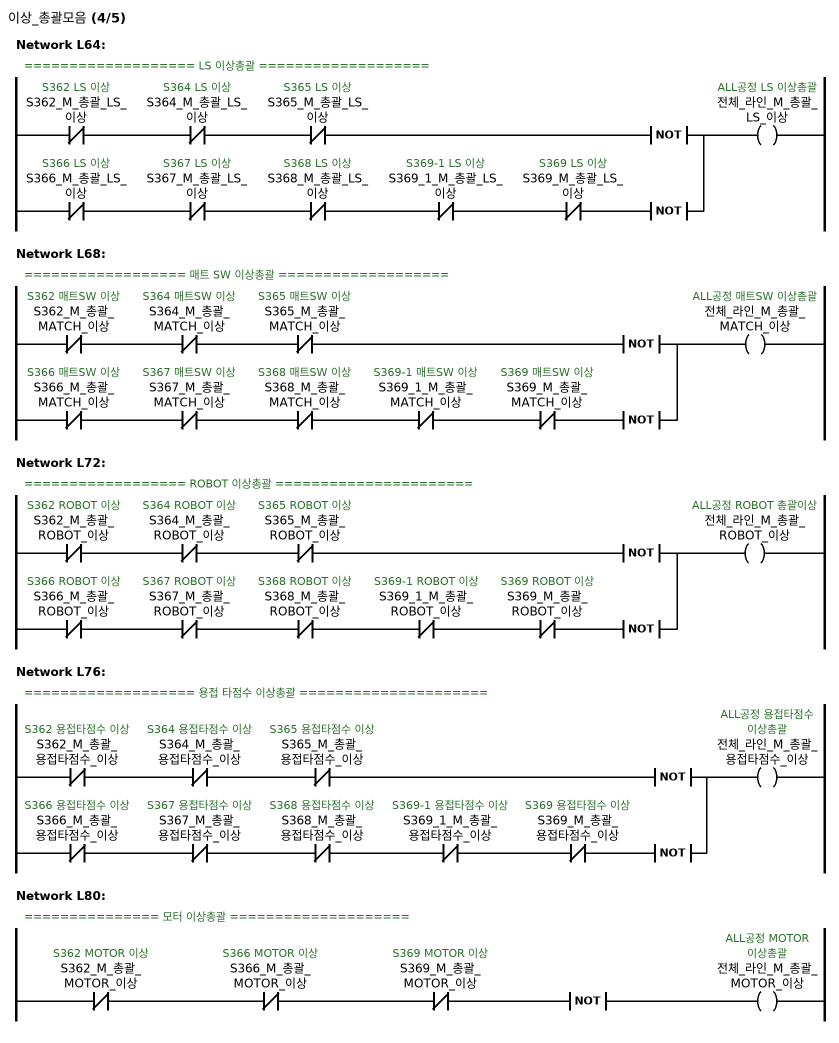
(* =================== LS 이상총괄 =================== *)
(* Rung L64 *)
전체_라인_M_총괄_LS_이상 := NOT (NOT S362_M_총괄_LS_이상 AND NOT S364_M_총괄_LS_이상 AND NOT S365_M_총괄_LS_이상) OR NOT (NOT S366_M_총괄_LS_이상 AND NOT S367_M_총괄_LS_이상 AND NOT S368_M_총괄_LS_이상 AND NOT S369_1_M_총괄_LS_이상 AND NOT S369_M_총괄_LS_이상);
(* ================== 매트 SW 이상총괄 =================== *)
(* Rung L68 *)
전체_라인_M_총괄_MATCH_이상 := NOT (NOT S362_M_총괄_MATCH_이상 AND NOT S364_M_총괄_MATCH_이상 AND NOT S365_M_총괄_MATCH_이상) OR NOT (NOT S366_M_총괄_MATCH_이상 AND NOT S367_M_총괄_MATCH_이상 AND NOT S368_M_총괄_MATCH_이상 AND NOT S369_1_M_총괄_MATCH_이상 AND NOT S369_M_총괄_MATCH_이상);
(* ================== ROBOT 이상총괄 ====================== *)
(* Rung L72 *)
전체_라인_M_총괄_ROBOT_이상 := NOT (NOT S362_M_총괄_ROBOT_이상 AND NOT S364_M_총괄_ROBOT_이상 AND NOT S365_M_총괄_ROBOT_이상) OR NOT (NOT S366_M_총괄_ROBOT_이상 AND NOT S367_M_총괄_ROBOT_이상 AND NOT S368_M_총괄_ROBOT_이상 AND NOT S369_1_M_총괄_ROBOT_이상 AND NOT S369_M_총괄_ROBOT_이상);
(* =================== 용접 타점수 이상총괄 ===================== *)
(* Rung L76 *)
전체_라인_M_총괄_용접타점수_이상 := NOT (NOT S362_M_총괄_용접타점수_이상 AND NOT S364_M_총괄_용접타점수_이상 AND NOT S365_M_총괄_용접타점수_이상) OR NOT (NOT S366_M_총괄_용접타점수_이상 AND NOT S367_M_총괄_용접타점수_이상 AND NOT S368_M_총괄_용접타점수_이상 AND NOT S369_1_M_총괄_용접타점수_이상 AND NOT S369_M_총괄_용접타점수_이상);
(* =============== 모터 이상총괄 ==================== *)
(* Rung L80 *)
전체_라인_M_총괄_MOTOR_이상 := NOT (NOT S362_M_총괄_MOTOR_이상 AND NOT S366_M_총괄_MOTOR_이상 AND NOT S369_M_총괄_MOTOR_이상);

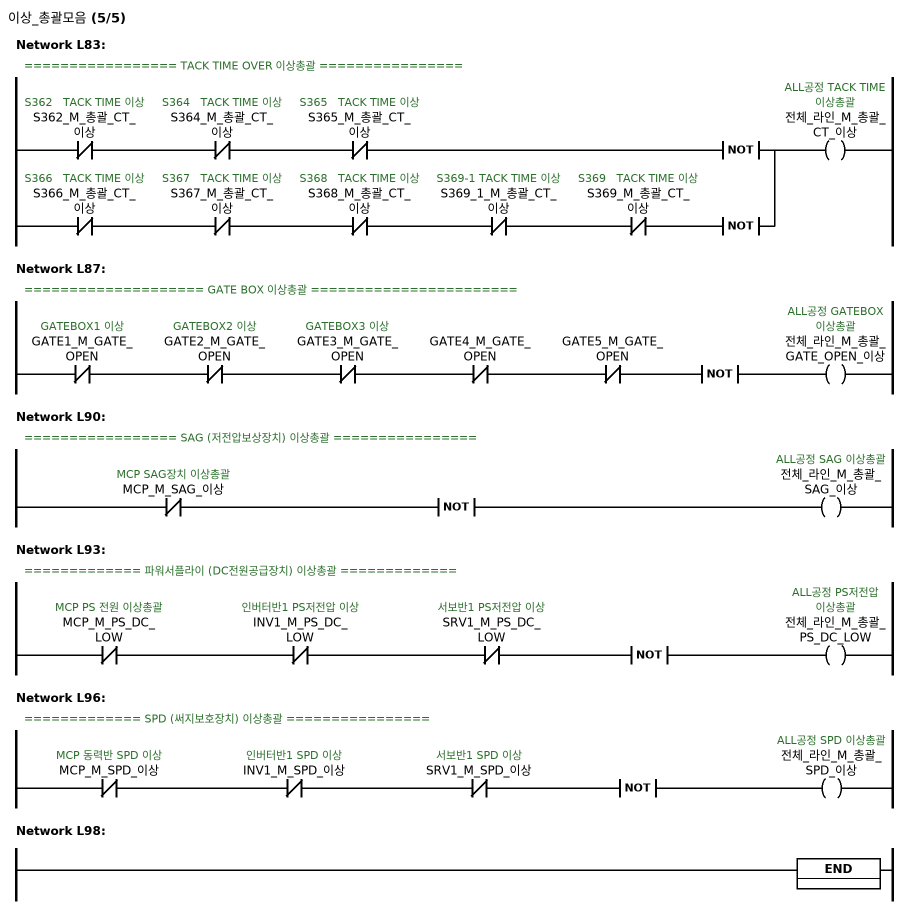
(* ================= TACK TIME OVER 이상총괄 ================ *)
(* Rung L83 *)
전체_라인_M_총괄_CT_이상 := NOT (NOT S362_M_총괄_CT_이상 AND NOT S364_M_총괄_CT_이상 AND NOT S365_M_총괄_CT_이상) OR NOT (NOT S366_M_총괄_CT_이상 AND NOT S367_M_총괄_CT_이상 AND NOT S368_M_총괄_CT_이상 AND NOT S369_1_M_총괄_CT_이상 AND NOT S369_M_총괄_CT_이상);
(* ==================== GATE BOX 이상총괄 ======================= *)
(* Rung L87 *)
전체_라인_M_총괄_GATE_OPEN_이상 := NOT (NOT GATE1_M_GATE_OPEN AND NOT GATE2_M_GATE_OPEN AND NOT GATE3_M_GATE_OPEN AND NOT GATE4_M_GATE_OPEN AND NOT GATE5_M_GATE_OPEN);
(* ================= SAG (저전압보상장치) 이상총괄 ================ *)
(* Rung L90 *)
전체_라인_M_총괄_SAG_이상 := MCP_M_SAG_이상;
(* ============= 파워서플라이 (DC전원공급장치) 이상총괄 ============= *)
(* Rung L93 *)
전체_라인_M_총괄_PS_DC_LOW := NOT (NOT MCP_M_PS_DC_LOW AND NOT INV1_M_PS_DC_LOW AND NOT SRV1_M_PS_DC_LOW);
(* ============= SPD (써지보호장치) 이상총괄 ================ *)
(* Rung L96 *)
전체_라인_M_총괄_SPD_이상 := NOT (NOT MCP_M_SPD_이상 AND NOT INV1_M_SPD_이상 AND NOT SRV1_M_SPD_이상);
(* Rung L98 *)
END();
END_PROGRAM

PROGRAM 이상_MCP (* task: 스캔 프로그램 *)
VAR_EXTERNAL RETAIN
    ALWAYS_OFF : BOOL; (* AT %MW3.0 *) (* 항시 OFF *)
    INV1_M_CP_OFF_이상 : BOOL; (* AT %MW355.3 *) (* 인버터반1 CP OFF 이상 *)
    INV1_M_PS_DC_LOW : BOOL; (* AT %MW355.2 *) (* 인버터반1 PS저전압 이상 *)
    INV1_M_SPD_이상 : BOOL; (* AT %MW355.1 *) (* 인버터반1 SPD 이상 *)
    INV1_M_총괄_이상 : BOOL; (* AT %MW355.0 *) (* INV1_M_총괄_이상 *)
    INV1_M_통신_이상 : BOOL; (* AT %MW355.4 *) (* 인버터반1 통신이상 *)
    MCP_M_CP_OFF_이상 : BOOL; (* AT %MW351.0 *) (* MCP CP OFF 이상총괄 *)
    MCP_M_DISPLAY_CP_TRIP : BOOL; (* AT %MW351.6 *) (* MCP 출력전원 CP OFF 이상 *)
    MCP_M_HUB_CP_TRIP : BOOL; (* AT %MW351.1 *) (* MCP PS전원 CP OFF 이상 *)
    MCP_M_INPUT_CP_TRIP : BOOL; (* AT %MW351.3 *) (* MCP HUB전원  CP OFF 이상 *)
    MCP_M_OUTPUT_CP_TRIP : BOOL; (* AT %MW351.4 *) (* MCP 통신모듈 전원 CP OFF 이상 *)
    MCP_M_OUTPUT_MC_이상 : BOOL; (* AT %MW354.8 *) (* MCP 운전준비 MC 이상 *)
    MCP_M_PROFI_PWR_CP_TRIP : BOOL; (* AT %MW351.5 *) (* MCP 입력전원 CP OFF 이상 *)
    MCP_M_PS1_DC_LOW : BOOL; (* AT %MW353.1 *) (* MCP PS1 전원 이상 *)
    MCP_M_PS2_DC_LOW : BOOL; (* AT %MW353.2 *) (* MCP PS2 전원 이상 *)
    MCP_M_PS3_DC_LOW : BOOL; (* AT %MW353.3 *) (* MCP PS3 전원 이상 *)
    MCP_M_PS4_DC_LOW : BOOL; (* AT %MW353.4 *) (* MCP PS4 전원 이상 *)
    MCP_M_PS_DC_LOW : BOOL; (* AT %MW353.0 *) (* MCP PS 전원 이상총괄 *)
    MCP_M_SAG1_1_이상 : BOOL; (* AT %MW352.1 *) (* MCP SAG장치 이상 *)
    MCP_M_SAG_이상 : BOOL; (* AT %MW352.0 *) (* MCP SAG장치 이상총괄 *)
    MCP_M_SPD_이상 : BOOL; (* AT %MW354.0 *) (* MCP 동력반 SPD 이상 *)
    MCP_M_이상_리셋 : BOOL; (* AT %MW350.4 *) (* MCP PB 이상리셋 *)
    MCP_M_총괄_이상 : BOOL; (* AT %MW302.0 *)
    MCP_M_통신_CP_TRIP : BOOL; (* AT %MW351.2 *) (* MCP   HMI전원  CP OFF 이상 *)
    MCP_M_통신_이상 : BOOL; (* AT %MW352.8 *) (* MCP 통신이상 *)
    SRV1_M_CP_OFF_이상 : BOOL; (* AT %MW356.3 *) (* 서보반1 CP OFF 이상 *)
    SRV1_M_PS_DC_LOW : BOOL; (* AT %MW356.2 *) (* 서보반1 PS저전압 이상 *)
    SRV1_M_SPD_이상 : BOOL; (* AT %MW356.1 *) (* 서보반1 SPD 이상 *)
    SRV1_M_총괄_이상 : BOOL; (* AT %MW356.0 *) (* SRV1_M_총괄_이상 *)
    SRV1_M_통신_이상 : BOOL; (* AT %MW356.4 *) (* SERVO반1 통신이상 *)
    전체_M_이상_리셋 : BOOL; (* AT %MW308.2 *) (* ALL공정 PB 이상리셋 *)
END_VAR
VAR_EXTERNAL
    EGIS_ON : BOOL; (* 항시ON (임시용) *)
    MCP_DISPLAY_CP_TRIP : BOOL; (* AT %MW87632.5 *) (* MCP 출력전원 CP TRIP *)
    MCP_HUB_CP_TRIP : BOOL; (* AT %MW87632.0 *) (* MCP PS1전원  CP TRIP *)
    MCP_INPUT_PWR_CP_TRIP : BOOL; (* AT %MW87632.2 *) (* MCP HUB전원  CP TRIP *)
    MCP_OUTPUT_PWR_CP1_TRIP : BOOL; (* AT %MW87632.3 *) (* MCP 통신모듈 전원 CP TRIP *)
    MCP_OUTPUT_PWR_CP2_TRIP : BOOL; (* AT %MW87632.4 *) (* MCP 입력전원 CP TRIP *)
    MCP_PS1_DC_OK : BOOL; (* AT %MW87631.12 *) (* MCP PS1 전원 정상 *)
    MCP_PS2_DC_OK : BOOL; (* AT %MW87631.13 *) (* MCP PS2 전원 정상 *)
    MCP_PS3_DC_OK : BOOL; (* AT %MW87631.14 *) (* MCP PS3 전원 정상 *)
    MCP_PS4_DC_OK : BOOL; (* AT %MW87631.15 *) (* MCP PS4 전원 정상 *)
    MCP_SAFTY_MC_ON : BOOL; (* AT %MW87632.9 *) (* MCP 운전준비 MC 보조접점 *)
    MCP_운전준비_MC_ON : BOOL; (* AT %MW97636.0 *) (* MCP 운전준비 MC ON *)
    MCP_통신_CP_TRIP : BOOL; (* AT %MW87632.1 *) (* MCP HMI전원  CP TRIP *)
    PWR_SAG1_DSUB1_NOMAL1 : BOOL; (* AT %MW87631.10 *) (* MCP SAG장치 정상 *)
    PWR_SAG1_DSUB8_NOMAL2 : BOOL; (* AT %MW87631.11 *) (* MCP SAG장치 이상 *)
    PWR_SPD1_NOMAL : BOOL; (* AT %MW87631.8 *) (* MCP 동력반 SPD 정상 *)
    S362_6_INV_BRAKE_CP_OFF : BOOL; (* AT %MW85013.13 *) (* S362_6_INV_BRAKE_CP_OFF *)
    S362_6_INV_DC_CP_TRIP : BOOL; (* AT %MW85013.12 *) (* S362_6_INV_DC_CP_TRIP *)
    S362_6_INV_PS1_DC_OK : BOOL; (* AT %MW85013.14 *) (* S362_6_INV_PS1_DC_OK *)
    S362_6_INV_SPD_NOMAL : BOOL; (* AT %MW85013.15 *) (* S362_6_INV_SPD_NOMAL *)
    S362_6_INV_제어_CP_OFF : BOOL; (* AT %MW85013.11 *) (* S362_6_INV_제어_CP_OFF *)
    SERVO_PNL_SPD_NOMAL : BOOL; (* AT %MW85023.14 *) (* SERVO_PNL_SPD_NOMAL *)
    SERVO_PS1_1_DC_OK : BOOL; (* AT %MW85023.12 *) (* SERVO_PS1_1_DC_OK *)
    SERVO_PS1_2_DC_OK : BOOL; (* AT %MW85023.13 *) (* SERVO_PS1_2_DC_OK *)
    SERVO_PS_CP_TRIP : BOOL; (* AT %MW85023.15 *) (* SERVO_PS_CP_TRIP *)
    _0007_EB63_CFG_ER : BOOL; (* AT %MW187088.0 *) (* EB 구성 에러 *)
    _0007_EB63_DEER : BOOL; (* AT %MW187088.1 *) (* EB 운전 중 탈락 *)
    _0007_EB63_IO_DEER : BOOL; (* AT %MW187089.2 *) (* EB IO 탈락 에러 *)
    _0007_EB63_IO_TYER : BOOL; (* AT %MW187089.1 *) (* EB IO 타입 에러 *)
    _MW87632_06 : BOOL; (* AT %MW87632.6 *) (* MCP 출력전원 CP TRIP *)
    _MW87632_07 : BOOL; (* AT %MW87632.7 *) (* MCP PC랙전원 CP TRIP *)
    _MW87632_08 : BOOL; (* AT %MW87632.8 *) (* MCP 현황판 CP TRIP *)
END_VAR
VAR
    INST15 : TON;
    INST16 : TON;
    INST17 : TON;
    INST18 : TON;
    INST19 : TON;
    INST24 : TON;
    INST25 : TON;
    INST26 : TON;
    INST27 : TON;
END_VAR

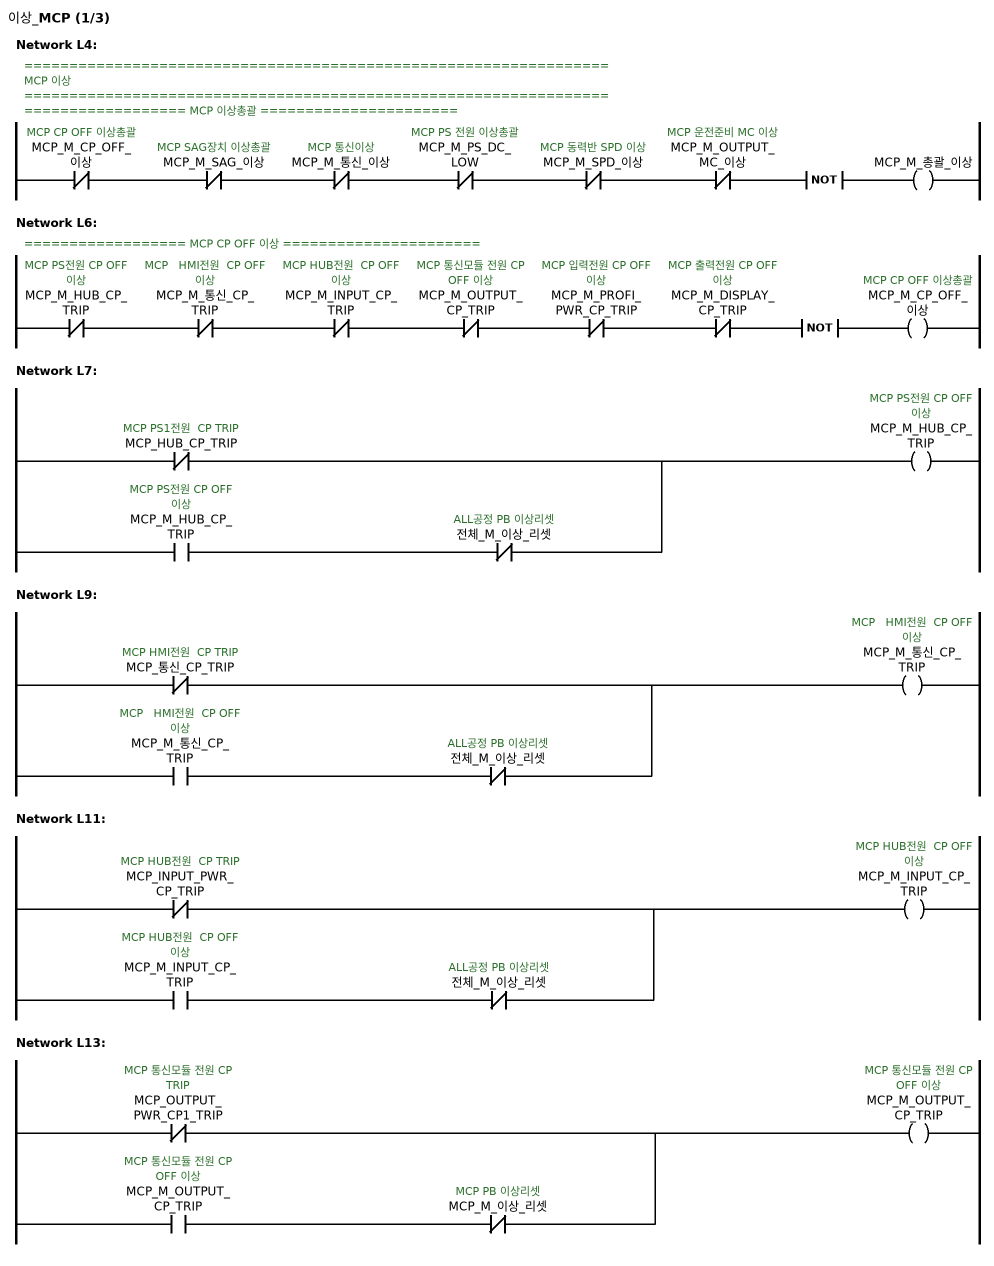
(* ================================================================= *)
(* MCP 이상 *)
(* ================================================================= *)
(* ================== MCP 이상총괄 ====================== *)
(* Rung L4 *)
MCP_M_총괄_이상 := NOT (NOT MCP_M_CP_OFF_이상 AND NOT MCP_M_SAG_이상 AND NOT MCP_M_통신_이상 AND NOT MCP_M_PS_DC_LOW AND NOT MCP_M_SPD_이상 AND NOT MCP_M_OUTPUT_MC_이상);
(* ================== MCP CP OFF 이상 ====================== *)
(* Rung L6 *)
MCP_M_CP_OFF_이상 := NOT (NOT MCP_M_HUB_CP_TRIP AND NOT MCP_M_통신_CP_TRIP AND NOT MCP_M_INPUT_CP_TRIP AND NOT MCP_M_OUTPUT_CP_TRIP AND NOT MCP_M_PROFI_PWR_CP_TRIP AND NOT MCP_M_DISPLAY_CP_TRIP);
(* Rung L7 *)
MCP_M_HUB_CP_TRIP := NOT MCP_HUB_CP_TRIP OR (MCP_M_HUB_CP_TRIP AND NOT 전체_M_이상_리셋);
(* Rung L9 *)
MCP_M_통신_CP_TRIP := NOT MCP_통신_CP_TRIP OR (MCP_M_통신_CP_TRIP AND NOT 전체_M_이상_리셋);
(* Rung L11 *)
MCP_M_INPUT_CP_TRIP := NOT MCP_INPUT_PWR_CP_TRIP OR (MCP_M_INPUT_CP_TRIP AND NOT 전체_M_이상_리셋);
(* Rung L13 *)
MCP_M_OUTPUT_CP_TRIP := NOT MCP_OUTPUT_PWR_CP1_TRIP OR (MCP_M_OUTPUT_CP_TRIP AND NOT MCP_M_이상_리셋);

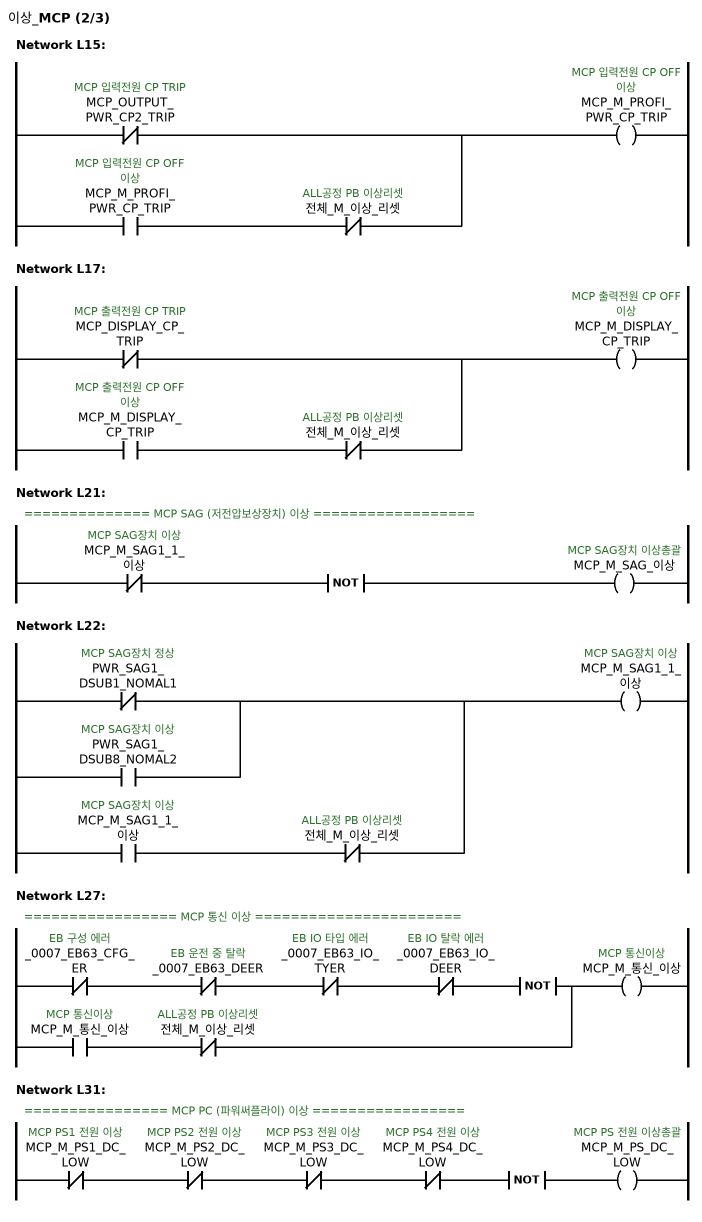
(* Rung L15 *)
MCP_M_PROFI_PWR_CP_TRIP := NOT MCP_OUTPUT_PWR_CP2_TRIP OR (MCP_M_PROFI_PWR_CP_TRIP AND NOT 전체_M_이상_리셋);
(* Rung L17 *)
MCP_M_DISPLAY_CP_TRIP := NOT MCP_DISPLAY_CP_TRIP OR (MCP_M_DISPLAY_CP_TRIP AND NOT 전체_M_이상_리셋);
(* ============== MCP SAG (저전압보상장치) 이상 ================== *)
(* Rung L21 *)
MCP_M_SAG_이상 := MCP_M_SAG1_1_이상;
(* Rung L22 *)
MCP_M_SAG1_1_이상 := NOT PWR_SAG1_DSUB1_NOMAL1 OR PWR_SAG1_DSUB8_NOMAL2 OR (MCP_M_SAG1_1_이상 AND NOT 전체_M_이상_리셋);
(* ================= MCP 통신 이상 ======================= *)
(* Rung L27 *)
MCP_M_통신_이상 := NOT (NOT _0007_EB63_CFG_ER AND NOT _0007_EB63_DEER AND NOT _0007_EB63_IO_TYER AND NOT _0007_EB63_IO_DEER) OR (MCP_M_통신_이상 AND NOT 전체_M_이상_리셋);
(* ================ MCP PC (파워써플라이) 이상 ================= *)
(* Rung L31 *)
MCP_M_PS_DC_LOW := NOT (NOT MCP_M_PS1_DC_LOW AND NOT MCP_M_PS2_DC_LOW AND NOT MCP_M_PS3_DC_LOW AND NOT MCP_M_PS4_DC_LOW);

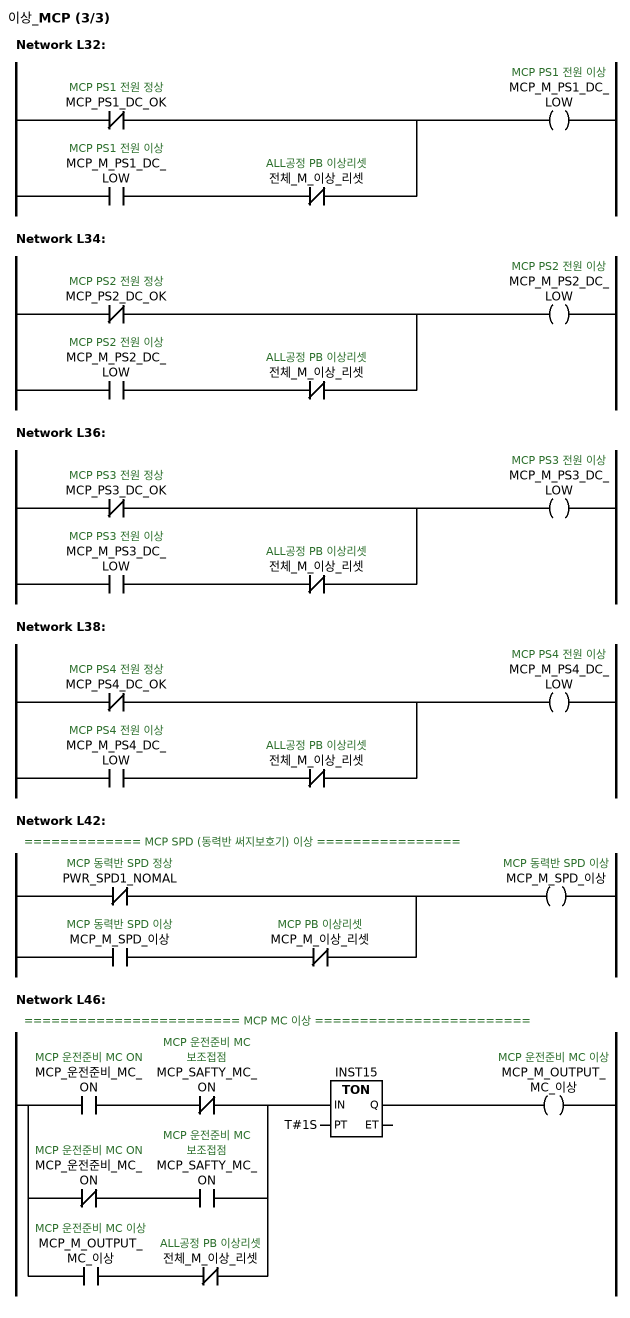
(* Rung L32 *)
MCP_M_PS1_DC_LOW := NOT MCP_PS1_DC_OK OR (MCP_M_PS1_DC_LOW AND NOT 전체_M_이상_리셋);
(* Rung L34 *)
MCP_M_PS2_DC_LOW := NOT MCP_PS2_DC_OK OR (MCP_M_PS2_DC_LOW AND NOT 전체_M_이상_리셋);
(* Rung L36 *)
MCP_M_PS3_DC_LOW := NOT MCP_PS3_DC_OK OR (MCP_M_PS3_DC_LOW AND NOT 전체_M_이상_리셋);
(* Rung L38 *)
MCP_M_PS4_DC_LOW := NOT MCP_PS4_DC_OK OR (MCP_M_PS4_DC_LOW AND NOT 전체_M_이상_리셋);
(* ============= MCP SPD (동력반 써지보호기) 이상 ================ *)
(* Rung L42 *)
MCP_M_SPD_이상 := NOT PWR_SPD1_NOMAL OR (MCP_M_SPD_이상 AND NOT MCP_M_이상_리셋);
(* ======================== MCP MC 이상 ======================== *)
(* Rung L46 *)
INST15(IN := (MCP_운전준비_MC_ON AND NOT MCP_SAFTY_MC_ON) OR (NOT MCP_운전준비_MC_ON AND MCP_SAFTY_MC_ON) OR (MCP_M_OUTPUT_MC_이상 AND NOT 전체_M_이상_리셋), PT := T#1S);
MCP_M_OUTPUT_MC_이상 := INST15.Q;
END_PROGRAM

PROGRAM 이상_인버터반 (* task: 스캔 프로그램 *)
VAR_EXTERNAL RETAIN
    ALWAYS_OFF : BOOL; (* AT %MW3.0 *) (* 항시 OFF *)
    INV1_M_CP_OFF_이상 : BOOL; (* AT %MW355.3 *) (* 인버터반1 CP OFF 이상 *)
    INV1_M_PS_DC_LOW : BOOL; (* AT %MW355.2 *) (* 인버터반1 PS저전압 이상 *)
    INV1_M_SPD_이상 : BOOL; (* AT %MW355.1 *) (* 인버터반1 SPD 이상 *)
    INV1_M_총괄_이상 : BOOL; (* AT %MW355.0 *) (* INV1_M_총괄_이상 *)
    INV1_M_통신_이상 : BOOL; (* AT %MW355.4 *) (* 인버터반1 통신이상 *)
    MCP_M_이상_리셋 : BOOL; (* AT %MW350.4 *) (* MCP PB 이상리셋 *)
    SRV1_M_CP_OFF_이상 : BOOL; (* AT %MW356.3 *) (* 서보반1 CP OFF 이상 *)
    SRV1_M_PS_DC_LOW : BOOL; (* AT %MW356.2 *) (* 서보반1 PS저전압 이상 *)
    SRV1_M_SPD_이상 : BOOL; (* AT %MW356.1 *) (* 서보반1 SPD 이상 *)
    SRV1_M_총괄_이상 : BOOL; (* AT %MW356.0 *) (* SRV1_M_총괄_이상 *)
    SRV1_M_통신_이상 : BOOL; (* AT %MW356.4 *) (* SERVO반1 통신이상 *)
END_VAR
VAR
    INST16 : TON;
    INST17 : TON;
    INST18 : TON;
    INST19 : TON;
    INST24 : TON;
    INST25 : TON;
    INST26 : TON;
    INST27 : TON;
END_VAR
VAR_EXTERNAL
    S362_6_INV_BRAKE_CP_OFF : BOOL; (* AT %MW85013.13 *) (* S362_6_INV_BRAKE_CP_OFF *)
    S362_6_INV_DC_CP_TRIP : BOOL; (* AT %MW85013.12 *) (* S362_6_INV_DC_CP_TRIP *)
    S362_6_INV_PS1_DC_OK : BOOL; (* AT %MW85013.14 *) (* S362_6_INV_PS1_DC_OK *)
    S362_6_INV_SPD_NOMAL : BOOL; (* AT %MW85013.15 *) (* S362_6_INV_SPD_NOMAL *)
    S362_6_INV_제어_CP_OFF : BOOL; (* AT %MW85013.11 *) (* S362_6_INV_제어_CP_OFF *)
    SERVO_PNL_SPD_NOMAL : BOOL; (* AT %MW85023.14 *) (* SERVO_PNL_SPD_NOMAL *)
    SERVO_PS1_1_DC_OK : BOOL; (* AT %MW85023.12 *) (* SERVO_PS1_1_DC_OK *)
    SERVO_PS1_2_DC_OK : BOOL; (* AT %MW85023.13 *) (* SERVO_PS1_2_DC_OK *)
    SERVO_PS_CP_TRIP : BOOL; (* AT %MW85023.15 *) (* SERVO_PS_CP_TRIP *)
    _0005_EB01_CFG_ER : BOOL; (* AT %MW185022.0 *) (* EB 구성 에러 *)
    _0005_EB01_DEER : BOOL; (* AT %MW185022.1 *) (* EB 운전 중 탈락 *)
    _0005_EB01_IO_DEER : BOOL; (* AT %MW185023.2 *) (* EB IO 탈락 에러 *)
    _0005_EB01_IO_TYER : BOOL; (* AT %MW185023.1 *) (* EB IO 타입 에러 *)
END_VAR

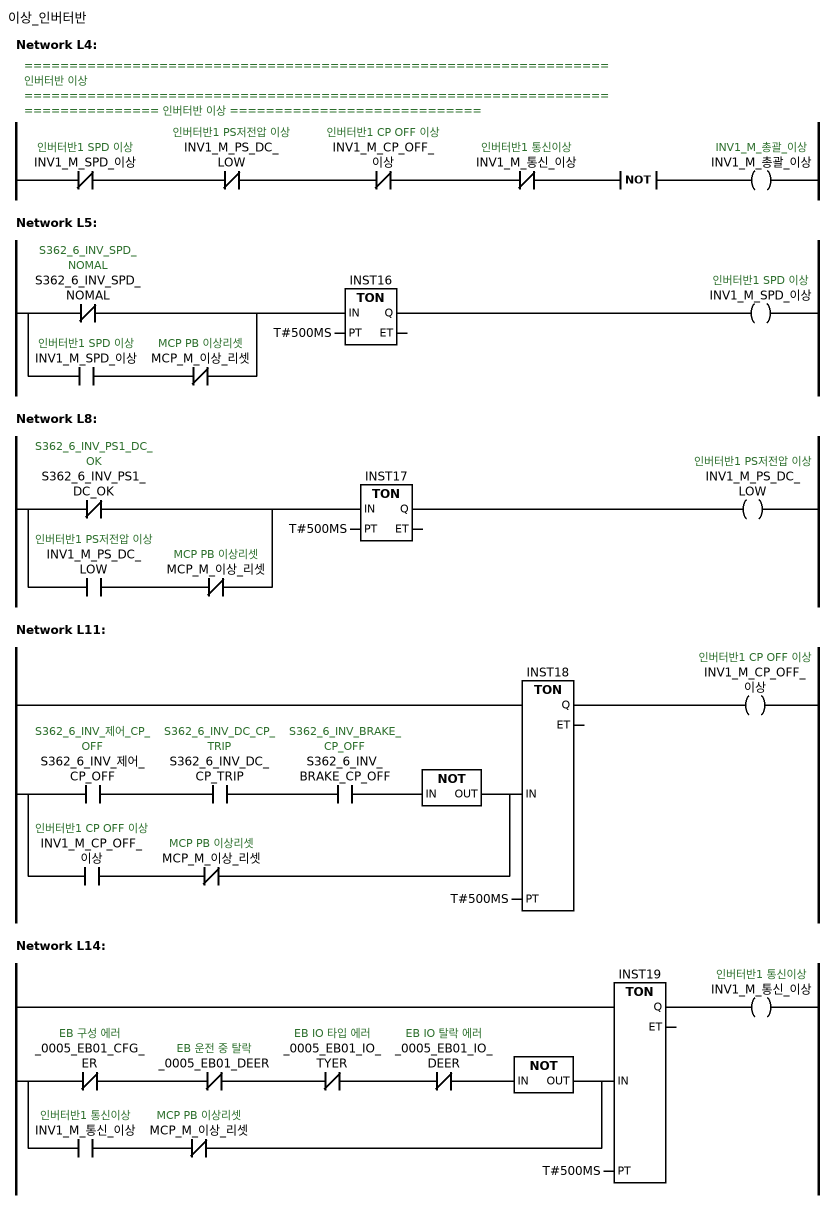
(* ================================================================= *)
(* 인버터반 이상 *)
(* ================================================================= *)
(* =============== 인버터반 이상 ============================ *)
(* Rung L4 *)
INV1_M_총괄_이상 := NOT (NOT INV1_M_SPD_이상 AND NOT INV1_M_PS_DC_LOW AND NOT INV1_M_CP_OFF_이상 AND NOT INV1_M_통신_이상);
(* Rung L5 *)
INST16(IN := NOT S362_6_INV_SPD_NOMAL OR (INV1_M_SPD_이상 AND NOT MCP_M_이상_리셋), PT := T#500MS);
INV1_M_SPD_이상 := INST16.Q;
(* Rung L8 *)
INST17(IN := NOT S362_6_INV_PS1_DC_OK OR (INV1_M_PS_DC_LOW AND NOT MCP_M_이상_리셋), PT := T#500MS);
INV1_M_PS_DC_LOW := INST17.Q;
(* Rung L11 *)
INST18(IN := (NOT (S362_6_INV_제어_CP_OFF AND S362_6_INV_DC_CP_TRIP AND S362_6_INV_BRAKE_CP_OFF)) OR (INV1_M_CP_OFF_이상 AND NOT MCP_M_이상_리셋), PT := T#500MS);
INV1_M_CP_OFF_이상 := INST18.Q;
(* Rung L14 *)
INST19(IN := (NOT (NOT _0005_EB01_CFG_ER AND NOT _0005_EB01_DEER AND NOT _0005_EB01_IO_TYER AND NOT _0005_EB01_IO_DEER)) OR (INV1_M_통신_이상 AND NOT MCP_M_이상_리셋), PT := T#500MS);
INV1_M_통신_이상 := INST19.Q;
END_PROGRAM

PROGRAM 이상_서보반 (* task: 스캔 프로그램 *)
VAR_EXTERNAL RETAIN
    ALWAYS_OFF : BOOL; (* AT %MW3.0 *) (* 항시 OFF *)
    MCP_M_이상_리셋 : BOOL; (* AT %MW350.4 *) (* MCP PB 이상리셋 *)
    SRV1_M_CP_OFF_이상 : BOOL; (* AT %MW356.3 *) (* 서보반1 CP OFF 이상 *)
    SRV1_M_PS_DC_LOW : BOOL; (* AT %MW356.2 *) (* 서보반1 PS저전압 이상 *)
    SRV1_M_SPD_이상 : BOOL; (* AT %MW356.1 *) (* 서보반1 SPD 이상 *)
    SRV1_M_총괄_이상 : BOOL; (* AT %MW356.0 *) (* SRV1_M_총괄_이상 *)
    SRV1_M_통신_이상 : BOOL; (* AT %MW356.4 *) (* SERVO반1 통신이상 *)
END_VAR
VAR
    INST24 : TON;
    INST25 : TON;
    INST26 : TON;
    INST27 : TON;
END_VAR
VAR_EXTERNAL
    SERVO_PNL_SPD_NOMAL : BOOL; (* AT %MW85023.14 *) (* SERVO_PNL_SPD_NOMAL *)
    SERVO_PS1_1_DC_OK : BOOL; (* AT %MW85023.12 *) (* SERVO_PS1_1_DC_OK *)
    SERVO_PS1_2_DC_OK : BOOL; (* AT %MW85023.13 *) (* SERVO_PS1_2_DC_OK *)
    SERVO_PS_CP_TRIP : BOOL; (* AT %MW85023.15 *) (* SERVO_PS_CP_TRIP *)
    _0005_EB01_CFG_ER : BOOL; (* AT %MW185022.0 *) (* EB 구성 에러 *)
    _0005_EB01_DEER : BOOL; (* AT %MW185022.1 *) (* EB 운전 중 탈락 *)
    _0005_EB01_IO_DEER : BOOL; (* AT %MW185023.2 *) (* EB IO 탈락 에러 *)
    _0005_EB01_IO_TYER : BOOL; (* AT %MW185023.1 *) (* EB IO 타입 에러 *)
    _0005_EB02_CFG_ER : BOOL; (* AT %MW185028.0 *) (* EB 구성 에러 *)
    _0005_EB02_DEER : BOOL; (* AT %MW185028.1 *) (* EB 운전 중 탈락 *)
    _0005_EB02_IO_DEER : BOOL; (* AT %MW185029.2 *) (* EB IO 탈락 에러 *)
    _0005_EB02_IO_TYER : BOOL; (* AT %MW185029.1 *) (* EB IO 타입 에러 *)
END_VAR

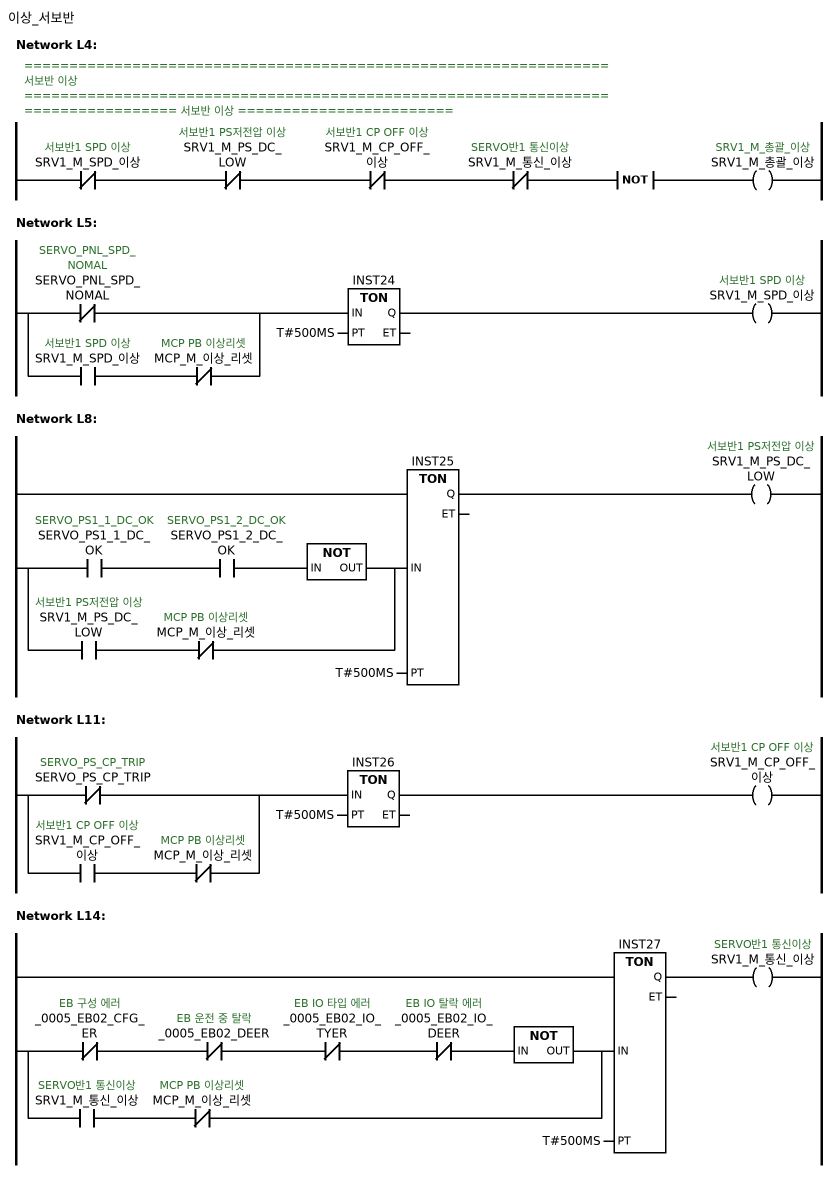
(* ================================================================= *)
(* 서보반 이상 *)
(* ================================================================= *)
(* ================= 서보반 이상 ======================== *)
(* Rung L4 *)
SRV1_M_총괄_이상 := NOT (NOT SRV1_M_SPD_이상 AND NOT SRV1_M_PS_DC_LOW AND NOT SRV1_M_CP_OFF_이상 AND NOT SRV1_M_통신_이상);
(* Rung L5 *)
INST24(IN := NOT SERVO_PNL_SPD_NOMAL OR (SRV1_M_SPD_이상 AND NOT MCP_M_이상_리셋), PT := T#500MS);
SRV1_M_SPD_이상 := INST24.Q;
(* Rung L8 *)
INST25(IN := (NOT (SERVO_PS1_1_DC_OK AND SERVO_PS1_2_DC_OK)) OR (SRV1_M_PS_DC_LOW AND NOT MCP_M_이상_리셋), PT := T#500MS);
SRV1_M_PS_DC_LOW := INST25.Q;
(* Rung L11 *)
INST26(IN := NOT SERVO_PS_CP_TRIP OR (SRV1_M_CP_OFF_이상 AND NOT MCP_M_이상_리셋), PT := T#500MS);
SRV1_M_CP_OFF_이상 := INST26.Q;
(* Rung L14 *)
INST27(IN := (NOT (NOT _0005_EB02_CFG_ER AND NOT _0005_EB02_DEER AND NOT _0005_EB02_IO_TYER AND NOT _0005_EB02_IO_DEER)) OR (SRV1_M_통신_이상 AND NOT MCP_M_이상_리셋), PT := T#500MS);
SRV1_M_통신_이상 := INST27.Q;
END_PROGRAM

PROGRAM 비상정지 (* task: 스캔 프로그램 *)
VAR_EXTERNAL RETAIN
    ALWAYS_OFF : BOOL; (* AT %MW3.0 *) (* 항시 OFF *)
    ALWAYS_ON : BOOL; (* AT %MW3.1 *) (* 항시 ON *)
    GATE1_M_EMSTOP : BOOL; (* AT %MW400.7 *) (* GATE1 비상정지 이상 *)
    GATE1_M_GATE_CLOSE : BOOL; (* AT %MW400.3 *) (* GATE1_M_GATE_CLOSE *)
    GATE1_M_비상정지_정상 : BOOL; (* AT %MW400.4 *)
    GATE2_M_EMSTOP : BOOL; (* AT %MW401.7 *) (* GATE2 비상정지 이상 *)
    GATE2_M_GATE_CLOSE : BOOL; (* AT %MW401.3 *) (* GATE2_M_GATE_CLOSE *)
    GATE2_M_비상정지_정상 : BOOL; (* AT %MW401.4 *)
    GATE3_M_EMSTOP : BOOL; (* AT %MW402.7 *) (* GATE3 비상정지 이상 *)
    GATE3_M_GATE_CLOSE : BOOL; (* AT %MW402.3 *) (* GATE3_M_GATE_CLOSE *)
    GATE3_M_비상정지_정상 : BOOL; (* AT %MW402.4 *)
    GATE4_M_EMSTOP : BOOL; (* AT %MW403.7 *)
    GATE4_M_GATE_CLOSE : BOOL; (* AT %MW403.3 *)
    GATE4_M_비상정지_정상 : BOOL; (* AT %MW403.4 *)
    GATE5_M_EMSTOP : BOOL; (* AT %MW404.7 *)
    GATE5_M_GATE_CLOSE : BOOL; (* AT %MW404.3 *)
    GATE5_M_비상정지_정상 : BOOL; (* AT %MW404.4 *)
    HOP1_M_EM_STOP_정상 : BOOL; (* AT %MW360.8 *)
    HOP1_M_비상정지 : BOOL; (* AT %MW360.7 *) (* HOP1 비상정지 이상 *)
    MCP_M_비상정지 : BOOL; (* AT %MW350.7 *) (* MCP 비상정지 이상 *)
    MCP_M_비상정지_정상 : BOOL; (* AT %MW350.8 *)
    MCP_M_이상_리셋 : BOOL; (* AT %MW350.4 *) (* MCP PB 이상리셋 *)
    S362_M_AOP_비상정지_이상 : BOOL; (* AT %MW1011.0 *) (* S362_M_AOP_비상정지_이상 *)
    S362_M_OP_ESTOP_NORMAL : BOOL; (* AT %MW1007.1 *) (* S362_M_OP_ESTOP_NORMAL *)
    S362_M_총괄_비상정지_이상 : BOOL; (* AT %MW1009.1 *) (* S362_M_총괄_비상정지_이상 *)
    S364_M_AOP_비상정지_이상 : BOOL; (* AT %MW2011.0 *) (* S364_M_AOP_비상정지_이상 *)
    S364_M_OP_ESTOP_NORMAL : BOOL; (* AT %MW2007.1 *) (* S364_M_OP_ESTOP_NORMAL *)
    S364_M_총괄_비상정지_이상 : BOOL; (* AT %MW2009.1 *) (* S364_M_총괄_비상정지_이상 *)
    S365_M_총괄_비상정지_이상 : BOOL; (* AT %MW2509.1 *) (* S365_M_총괄_비상정지_이상 *)
    S366_M_총괄_비상정지_이상 : BOOL; (* AT %MW3009.1 *) (* S366_M_총괄_비상정지_이상 *)
    S367_M_총괄_비상정지_이상 : BOOL; (* AT %MW3509.1 *) (* S367_M_총괄_비상정지_이상 *)
    S368_M_총괄_비상정지_이상 : BOOL; (* AT %MW4009.1 *) (* S368_M_총괄_비상정지_이상 *)
    S369_M_총괄_비상정지_이상 : BOOL; (* AT %MW5009.1 *) (* S369_M_총괄_비상정지_이상 *)
    전체_M_GATE_비상정지_정상 : BOOL; (* AT %MW308.4 *) (* 전체 M GATE 비상정지 정상 *)
    전체_M_이상_리셋 : BOOL; (* AT %MW308.2 *) (* ALL공정 PB 이상리셋 *)
    전체_OP_M_총괄_비상정지_정상 : BOOL; (* AT %MW304.2 *)
    전체_공정_M_총괄_비상정지_정상 : BOOL; (* AT %MW304.1 *)
    전체_라인_M_총괄_비상정지_정상 : BOOL; (* AT %MW304.0 *)
END_VAR
VAR_EXTERNAL
    GB1_EPB_비상정지1 : BOOL; (* AT %MW87012.0 *) (* GB1_EPB_비상정지1 *)
    GB1_EPB_비상정지2 : BOOL; (* AT %MW87012.1 *) (* GB1_EPB_비상정지2 *)
    GB2_EPB_비상정지1 : BOOL; (* AT %MW87022.0 *) (* GB2_EPB_비상정지1 *)
    GB2_EPB_비상정지2 : BOOL; (* AT %MW87022.1 *) (* GB2_EPB_비상정지2 *)
    GB3_EPB_비상정지1 : BOOL; (* AT %MW87032.0 *) (* GB3_EPB_비상정지1 *)
    GB3_EPB_비상정지2 : BOOL; (* AT %MW87032.1 *) (* GB3_EPB_비상정지2 *)
    GB4_EPB_비상정지1 : BOOL; (* AT %MW87112.0 *) (* GB4 EPB 비상정지1 *)
    GB4_EPB_비상정지2 : BOOL; (* AT %MW87112.1 *) (* GB4 EPB 비상정지2 *)
    GB5_EPB_비상정지1 : BOOL; (* AT %MW87122.0 *) (* GB5 EPB 비상정지1 *)
    GB5_EPB_비상정지2 : BOOL; (* AT %MW87122.1 *) (* GB5 EPB 비상정지2 *)
    HOP_EPB_비상정지1 : BOOL; (* AT %MW87503.8 *) (* HOP_EPB_비상정지1 *)
    HOP_EPB_비상정지2 : BOOL; (* AT %MW87503.9 *) (* HOP_EPB_비상정지2 *)
    MCP_EPB_비상정지1 : BOOL; (* AT %MW87635.0 *) (* MCP_EPB_비상정지1 *)
    MCP_EPB_비상정지2 : BOOL; (* AT %MW87635.1 *) (* MCP_EPB_비상정지2 *)
    R361_1_M_I_RB_비상정지 : BOOL; (* AT %MW20010.4 *) (* R361_1_M_I_RB_비상정지 *)
    R361_2_M_I_RB_비상정지 : BOOL; (* AT %MW20020.4 *) (* R361_2_M_I_RB_비상정지 *)
    R363_1_M_I_RB_비상정지 : BOOL; (* AT %MW20030.4 *) (* R363_1_M_I_RB_비상정지 *)
    R363_2_M_I_RB_비상정지 : BOOL; (* AT %MW20040.4 *) (* R363_2_M_I_RB_비상정지 *)
    R364_1_M_I_RB_비상정지 : BOOL; (* AT %MW20050.4 *) (* R364_1_M_I_RB_비상정지 *)
    R366_1_M_I_RB_비상정지 : BOOL; (* AT %MW20060.4 *) (* R366_1_M_I_RB_비상정지 *)
    R368_1_M_I_RB_비상정지 : BOOL; (* AT %MW20070.4 *) (* R368_1_M_I_RB_비상정지 *)
    R369_1_M_I_RB_비상정지 : BOOL; (* AT %MW20080.4 *) (* R369_1_M_I_RB_비상정지 *)
    R369_2_M_I_RB_비상정지 : BOOL; (* AT %MW20090.4 *) (* R369_2_M_I_RB_비상정지 *)
    S362_EPB_AX_비상정지1 : BOOL; (* AT %MW87105.0 *) (* S362_EPB_AX_비상정지1 *)
    S362_EPB_AX_비상정지2 : BOOL; (* AT %MW87105.1 *) (* S362_EPB_AX_비상정지2 *)
    S364_EPB_AX_비상정지1 : BOOL; (* AT %MW87155.0 *) (* S364_EPB_AX_비상정지1 *)
    S364_EPB_AX_비상정지2 : BOOL; (* AT %MW87155.1 *) (* S364_EPB_AX_비상정지2 *)
END_VAR

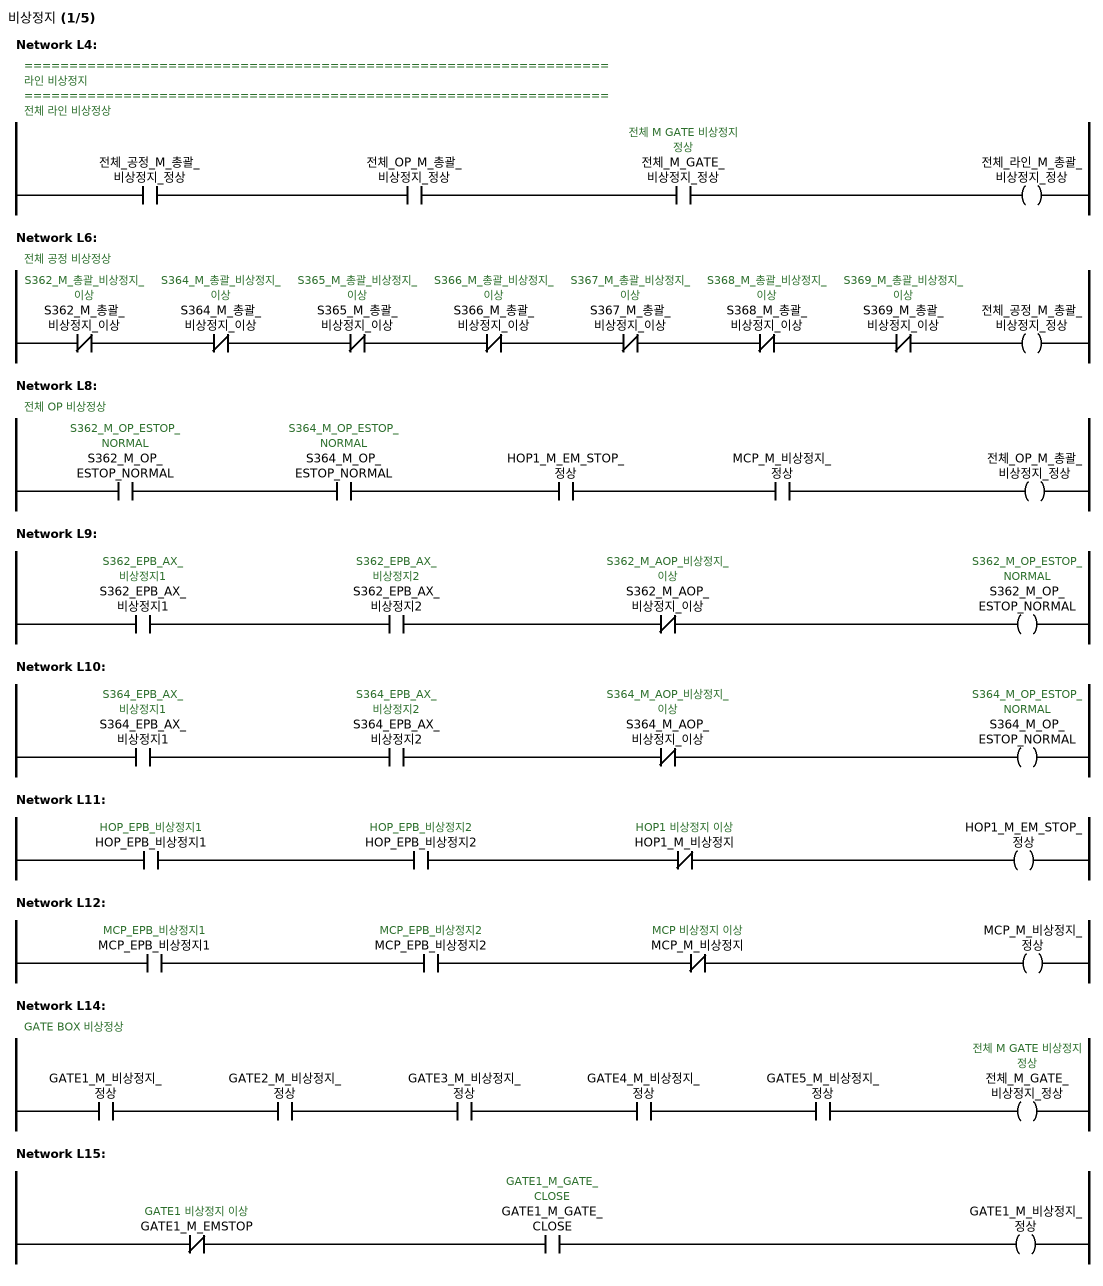
(* ================================================================= *)
(* 라인 비상정지 *)
(* ================================================================= *)
(* 전체 라인 비상정상 *)
(* Rung L4 *)
전체_라인_M_총괄_비상정지_정상 := 전체_공정_M_총괄_비상정지_정상 AND 전체_OP_M_총괄_비상정지_정상 AND 전체_M_GATE_비상정지_정상;
(* 전체 공정 비상정상 *)
(* Rung L6 *)
전체_공정_M_총괄_비상정지_정상 := NOT S362_M_총괄_비상정지_이상 AND NOT S364_M_총괄_비상정지_이상 AND NOT S365_M_총괄_비상정지_이상 AND NOT S366_M_총괄_비상정지_이상 AND NOT S367_M_총괄_비상정지_이상 AND NOT S368_M_총괄_비상정지_이상 AND NOT S369_M_총괄_비상정지_이상;
(* 전체 OP 비상정상 *)
(* Rung L8 *)
전체_OP_M_총괄_비상정지_정상 := S362_M_OP_ESTOP_NORMAL AND S364_M_OP_ESTOP_NORMAL AND HOP1_M_EM_STOP_정상 AND MCP_M_비상정지_정상;
(* Rung L9 *)
S362_M_OP_ESTOP_NORMAL := S362_EPB_AX_비상정지1 AND S362_EPB_AX_비상정지2 AND NOT S362_M_AOP_비상정지_이상;
(* Rung L10 *)
S364_M_OP_ESTOP_NORMAL := S364_EPB_AX_비상정지1 AND S364_EPB_AX_비상정지2 AND NOT S364_M_AOP_비상정지_이상;
(* Rung L11 *)
HOP1_M_EM_STOP_정상 := HOP_EPB_비상정지1 AND HOP_EPB_비상정지2 AND NOT HOP1_M_비상정지;
(* Rung L12 *)
MCP_M_비상정지_정상 := MCP_EPB_비상정지1 AND MCP_EPB_비상정지2 AND NOT MCP_M_비상정지;
(* GATE BOX 비상정상 *)
(* Rung L14 *)
전체_M_GATE_비상정지_정상 := GATE1_M_비상정지_정상 AND GATE2_M_비상정지_정상 AND GATE3_M_비상정지_정상 AND GATE4_M_비상정지_정상 AND GATE5_M_비상정지_정상;
(* Rung L15 *)
GATE1_M_비상정지_정상 := NOT GATE1_M_EMSTOP AND GATE1_M_GATE_CLOSE;

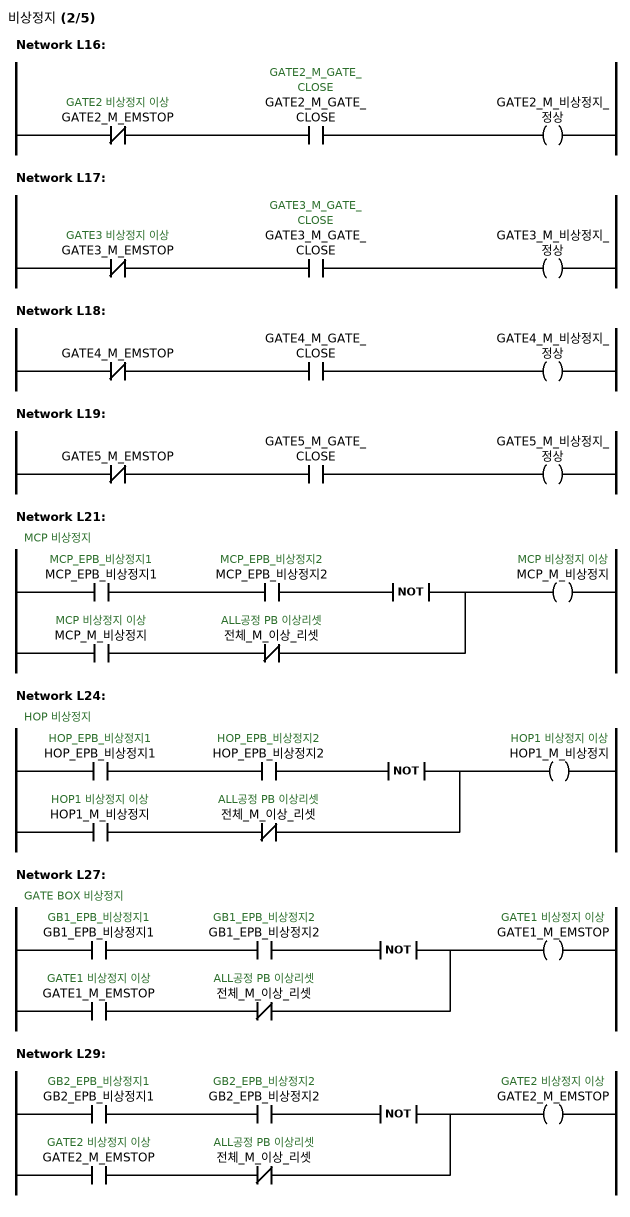
(* Rung L16 *)
GATE2_M_비상정지_정상 := NOT GATE2_M_EMSTOP AND GATE2_M_GATE_CLOSE;
(* Rung L17 *)
GATE3_M_비상정지_정상 := NOT GATE3_M_EMSTOP AND GATE3_M_GATE_CLOSE;
(* Rung L18 *)
GATE4_M_비상정지_정상 := NOT GATE4_M_EMSTOP AND GATE4_M_GATE_CLOSE;
(* Rung L19 *)
GATE5_M_비상정지_정상 := NOT GATE5_M_EMSTOP AND GATE5_M_GATE_CLOSE;
(* MCP 비상정지 *)
(* Rung L21 *)
MCP_M_비상정지 := NOT (MCP_EPB_비상정지1 AND MCP_EPB_비상정지2) OR (MCP_M_비상정지 AND NOT 전체_M_이상_리셋);
(* HOP 비상정지 *)
(* Rung L24 *)
HOP1_M_비상정지 := NOT (HOP_EPB_비상정지1 AND HOP_EPB_비상정지2) OR (HOP1_M_비상정지 AND NOT 전체_M_이상_리셋);
(* GATE BOX 비상정지 *)
(* Rung L27 *)
GATE1_M_EMSTOP := NOT (GB1_EPB_비상정지1 AND GB1_EPB_비상정지2) OR (GATE1_M_EMSTOP AND NOT 전체_M_이상_리셋);
(* Rung L29 *)
GATE2_M_EMSTOP := NOT (GB2_EPB_비상정지1 AND GB2_EPB_비상정지2) OR (GATE2_M_EMSTOP AND NOT 전체_M_이상_리셋);

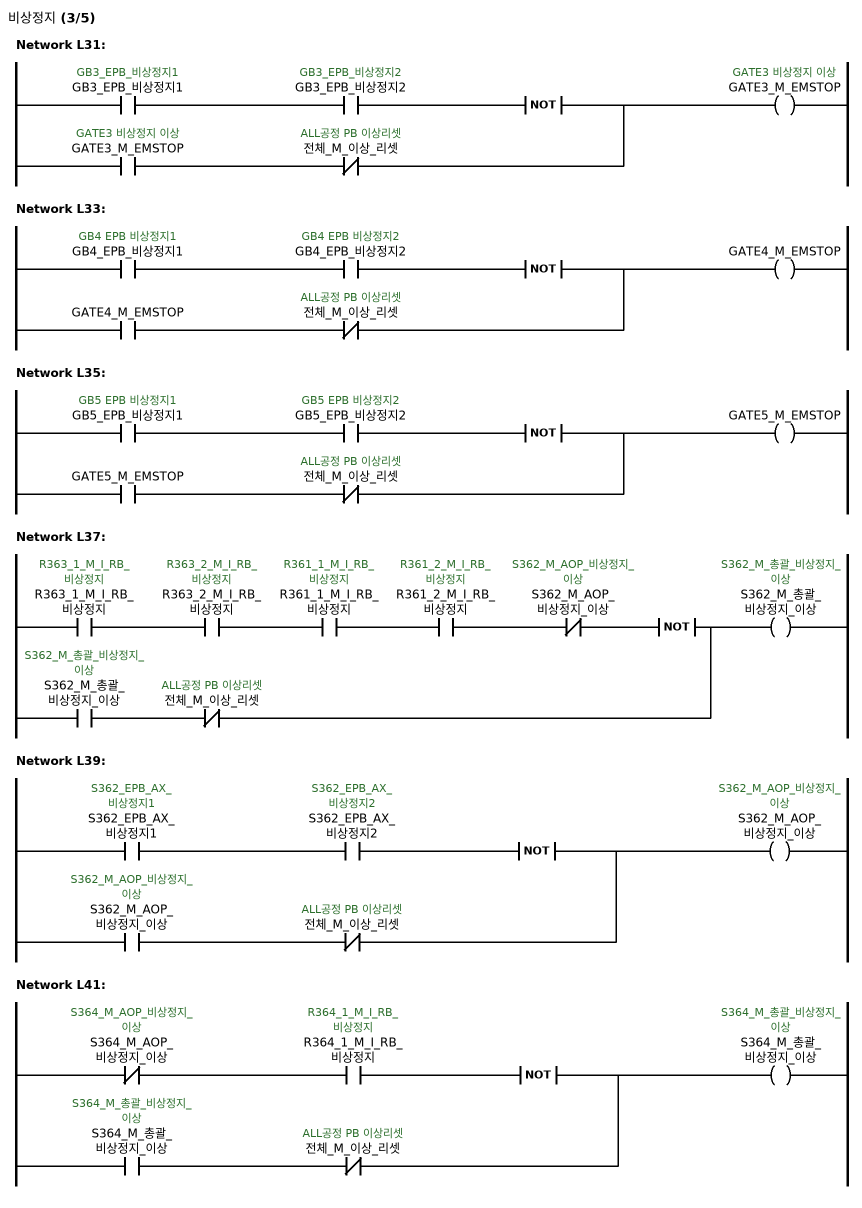
(* Rung L31 *)
GATE3_M_EMSTOP := NOT (GB3_EPB_비상정지1 AND GB3_EPB_비상정지2) OR (GATE3_M_EMSTOP AND NOT 전체_M_이상_리셋);
(* Rung L33 *)
GATE4_M_EMSTOP := NOT (GB4_EPB_비상정지1 AND GB4_EPB_비상정지2) OR (GATE4_M_EMSTOP AND NOT 전체_M_이상_리셋);
(* Rung L35 *)
GATE5_M_EMSTOP := NOT (GB5_EPB_비상정지1 AND GB5_EPB_비상정지2) OR (GATE5_M_EMSTOP AND NOT 전체_M_이상_리셋);
(* Rung L37 *)
S362_M_총괄_비상정지_이상 := NOT (R363_1_M_I_RB_비상정지 AND R363_2_M_I_RB_비상정지 AND R361_1_M_I_RB_비상정지 AND R361_2_M_I_RB_비상정지 AND NOT S362_M_AOP_비상정지_이상) OR (S362_M_총괄_비상정지_이상 AND NOT 전체_M_이상_리셋);
(* Rung L39 *)
S362_M_AOP_비상정지_이상 := NOT (S362_EPB_AX_비상정지1 AND S362_EPB_AX_비상정지2) OR (S362_M_AOP_비상정지_이상 AND NOT 전체_M_이상_리셋);
(* Rung L41 *)
S364_M_총괄_비상정지_이상 := NOT (NOT S364_M_AOP_비상정지_이상 AND R364_1_M_I_RB_비상정지) OR (S364_M_총괄_비상정지_이상 AND NOT 전체_M_이상_리셋);

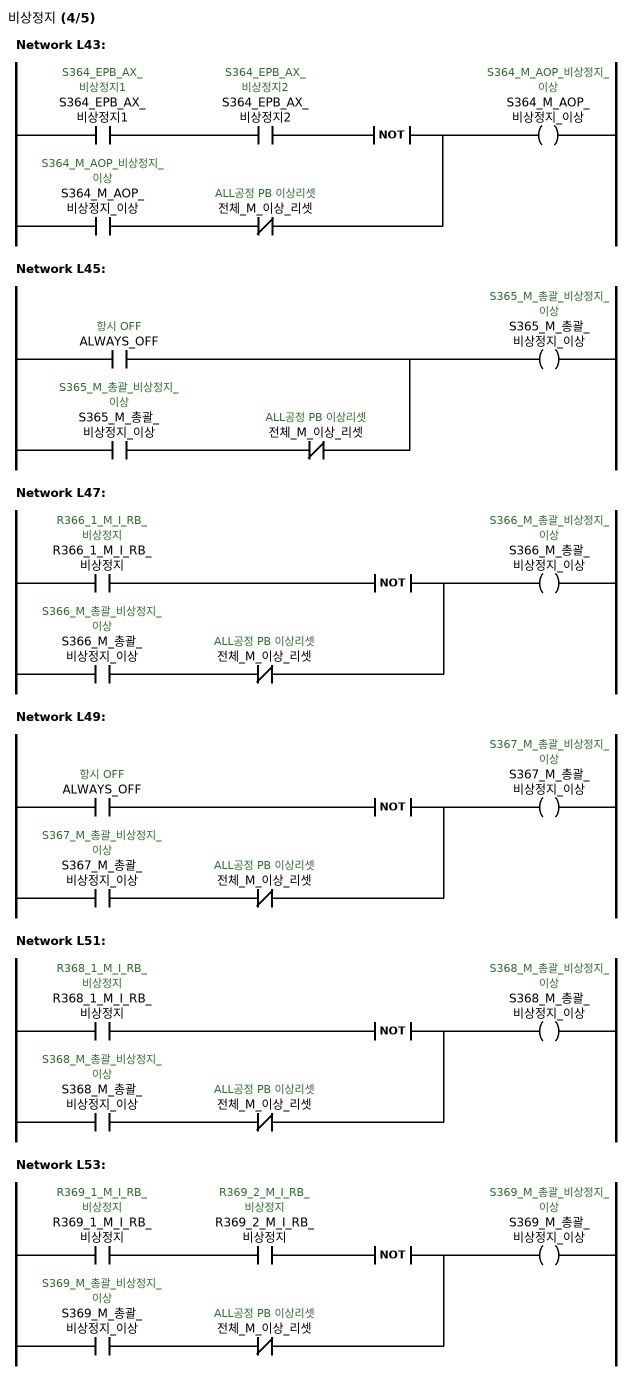
(* Rung L43 *)
S364_M_AOP_비상정지_이상 := NOT (S364_EPB_AX_비상정지1 AND S364_EPB_AX_비상정지2) OR (S364_M_AOP_비상정지_이상 AND NOT 전체_M_이상_리셋);
(* Rung L45 *)
S365_M_총괄_비상정지_이상 := ALWAYS_OFF OR (S365_M_총괄_비상정지_이상 AND NOT 전체_M_이상_리셋);
(* Rung L47 *)
S366_M_총괄_비상정지_이상 := NOT R366_1_M_I_RB_비상정지 OR (S366_M_총괄_비상정지_이상 AND NOT 전체_M_이상_리셋);
(* Rung L49 *)
S367_M_총괄_비상정지_이상 := NOT ALWAYS_OFF OR (S367_M_총괄_비상정지_이상 AND NOT 전체_M_이상_리셋);
(* Rung L51 *)
S368_M_총괄_비상정지_이상 := NOT R368_1_M_I_RB_비상정지 OR (S368_M_총괄_비상정지_이상 AND NOT 전체_M_이상_리셋);
(* Rung L53 *)
S369_M_총괄_비상정지_이상 := NOT (R369_1_M_I_RB_비상정지 AND R369_2_M_I_RB_비상정지) OR (S369_M_총괄_비상정지_이상 AND NOT 전체_M_이상_리셋);

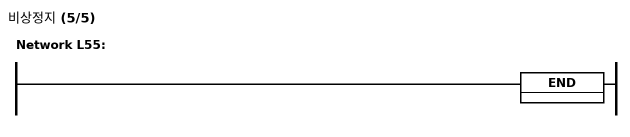
(* Rung L55 *)
END();
END_PROGRAM

PROGRAM ROOF_RACK_유틸리티 (* task: 스캔 프로그램 *)
VAR_EXTERNAL RETAIN
    HMI_M_선택_MOD_ROOF_RACK : BOOL; (* AT %MW6.1 *) (* HMI M 선택 MOD S363 *)
    HMI_M_선택_MOD_S362 : BOOL; (* AT %MW6.0 *) (* HMI M 선택 MOD S362 *)
    R361_1_M_SEQ : WORD; (* AT %MW10000 *) (* R361 1 M SEQ *)
    R361_1_M_공정_차종_유 : BOOL; (* S362_M_공정_차종_유 *)
    R361_1_M_차종1_AX : BOOL; (* AT %MW10001.0 *) (* R361 1 M 차종1 AX *)
    R361_1_M_차종1_B : BOOL; (* AT %MW10001.1 *) (* R361 1 M 차종1 B *)
    R361_1_M_차종1_C : BOOL; (* AT %MW10001.2 *) (* R361 1 M 차종1 C *)
    R361_1_M_차종1_D : BOOL; (* AT %MW10001.3 *) (* R361 1 M 차종1 D *)
    R361_1_M_차종1_E : BOOL; (* AT %MW10001.4 *) (* R361 1 M 차종1 E *)
    R361_1_M_차종1_F : BOOL; (* AT %MW10001.5 *) (* R361 1 M 차종1 F *)
    R361_1_M_차종1_G : BOOL; (* AT %MW10001.6 *) (* R361 1 M 차종1 G *)
    R361_1_M_차종1_H : BOOL; (* AT %MW10001.7 *) (* R361 1 M 차종1 H *)
    R361_1_M_차종2_3DR : BOOL; (* AT %MW10001.8 *) (* R361 1 M 차종2 3DR *)
    R361_1_M_차종2_4DR : BOOL; (* AT %MW10001.9 *) (* R361 1 M 차종2 4DR *)
    R361_1_M_차종2_5DR : BOOL; (* AT %MW10001.10 *) (* R361 1 M 차종2 5DR *)
    R361_1_M_차종2_SP1 : BOOL; (* AT %MW10001.12 *) (* R361 1 M 차종2 SP1 *)
    R361_1_M_차종2_SP2 : BOOL; (* AT %MW10001.13 *) (* R361 1 M 차종2 SP2 *)
    R361_1_M_차종2_WGN : BOOL; (* AT %MW10001.11 *) (* R361 1 M 차종2 WGN *)
    R361_1_M_차종3_LHD : BOOL; (* AT %MW10001.14 *) (* R361 1 M 차종3 LHD *)
    R361_1_M_차종3_RHD : BOOL; (* AT %MW10001.15 *) (* R361 1 M 차종3 RHD *)
    R361_1_M_차종4_EEC : BOOL; (* AT %MW10002.3 *) (* R361 1 M 차종4 EEC *)
    R361_1_M_차종4_SP1 : BOOL; (* AT %MW10002.8 *) (* R361 1 M 차종4 SP1 *)
    R361_1_M_차종4_SP2 : BOOL; (* AT %MW10002.9 *) (* R361 1 M 차종4 SP2 *)
    R361_1_M_차종4_SP3 : BOOL; (* AT %MW10002.11 *) (* R361 1 M 차종4 SP3 *)
    R361_1_M_차종4_SP4 : BOOL; (* AT %MW10002.12 *) (* R361 1 M 차종4 SP4 *)
    R361_1_M_차종4_SP5 : BOOL; (* AT %MW10002.13 *) (* R361 1 M 차종4 SP5 *)
    R361_1_M_차종4_SP6 : BOOL; (* AT %MW10002.14 *) (* R361 1 M 차종4 SP6 *)
    R361_1_M_차종4_SP7 : BOOL; (* AT %MW10002.15 *) (* R361 1 M 차종4 SP7 *)
    R361_1_M_차종4_내수 : BOOL; (* AT %MW10002.0 *) (* R361 1 M 차종4 내수 *)
    R361_1_M_차종4_러시아 : BOOL; (* AT %MW10002.10 *) (* R361 1 M 차종4 러시아 *)
    R361_1_M_차종4_북미 : BOOL; (* AT %MW10002.2 *) (* R361 1 M 차종4 북미 *)
    R361_1_M_차종4_브라질 : BOOL; (* AT %MW10002.7 *) (* R361 1 M 차종4 브라질 *)
    R361_1_M_차종4_수출 : BOOL; (* AT %MW10002.1 *) (* R361 1 M 차종4 수출 *)
    R361_1_M_차종4_중국 : BOOL; (* AT %MW10002.6 *) (* R361 1 M 차종4 중국 *)
    R361_1_M_차종4_중동 : BOOL; (* AT %MW10002.5 *) (* R361 1 M 차종4 중동 *)
    R361_1_M_차종4_호주 : BOOL; (* AT %MW10002.4 *) (* R361 1 M 차종4 호주 *)
    R361_1_M_차종5_AT : BOOL; (* AT %MW10003.1 *) (* R361 1 M 차종5 AT *)
    R361_1_M_차종5_MT : BOOL; (* AT %MW10003.0 *) (* R361 1 M 차종5 MT *)
    R361_1_M_차종5_SP1 : BOOL; (* AT %MW10003.2 *) (* R361 1 M 차종5 SP1 *)
    R361_1_M_차종6_DSROOF : BOOL; (* AT %MW10003.6 *) (* R361 1 M 차종6 DSROOF *)
    R361_1_M_차종6_SP1 : BOOL; (* AT %MW10003.7 *) (* R361 1 M 차종6 SP1 *)
    R361_1_M_차종6_썬루프 : BOOL; (* AT %MW10003.4 *) (* R361 1 M 차종6 썬루프 *)
    R361_1_M_차종6_일반루프 : BOOL; (* AT %MW10003.3 *) (* R361 1 M 차종6 일반루프 *)
    R361_1_M_차종6_파노라마루프 : BOOL; (* AT %MW10003.5 *) (* R361 1 M 차종6 파노라마루프 *)
    R361_1_M_차종7_DSL : BOOL; (* AT %MW10003.9 *) (* R361 1 M 차종7 DSL *)
    R361_1_M_차종7_GSL : BOOL; (* AT %MW10003.8 *) (* R361 1 M 차종7 GSL *)
    R361_1_M_차종7_SP1 : BOOL; (* AT %MW10003.10 *) (* R361 1 M 차종7 SP1 *)
    R361_1_M_차종7_SP2 : BOOL; (* AT %MW10003.11 *) (* R361 1 M 차종7 SP2 *)
    R361_1_M_차종7_SP3 : BOOL; (* AT %MW10003.12 *) (* R361 1 M 차종7 SP3 *)
    R361_1_M_차종7_SP4 : BOOL; (* AT %MW10003.13 *) (* R361 1 M 차종7 SP4 *)
    R361_1_M_차종7_SP5 : BOOL; (* AT %MW10003.14 *) (* R361 1 M 차종7 SP5 *)
    R361_1_M_차종7_SP6 : BOOL; (* AT %MW10003.15 *) (* R361 1 M 차종7 SP6 *)
    R361_1_M_차종8_2WD : BOOL; (* AT %MW10004.0 *) (* R361 1 M 차종8 2WD *)
    R361_1_M_차종8_4WD : BOOL; (* AT %MW10004.1 *) (* R361 1 M 차종8 4WD *)
    R361_1_M_차종8_SP1 : BOOL; (* AT %MW10004.2 *) (* R361 1 M 차종8 SP1 *)
    R361_1_M_차종9_MPI : BOOL; (* AT %MW10004.3 *) (* R361 1 M 차종9 MPI *)
    R361_1_M_차종9_SP1 : BOOL; (* AT %MW10004.5 *) (* R361 1 M 차종9 SP1 *)
    R361_1_M_차종9_SP10 : BOOL; (* AT %MW10004.14 *) (* R361 1 M 차종9 SP10 *)
    R361_1_M_차종9_SP11 : BOOL; (* AT %MW10004.15 *) (* R361 1 M 차종9 SP11 *)
    R361_1_M_차종9_SP2 : BOOL; (* AT %MW10004.6 *) (* R361 1 M 차종9 SP2 *)
    R361_1_M_차종9_SP3 : BOOL; (* AT %MW10004.7 *) (* R361 1 M 차종9 SP3 *)
    R361_1_M_차종9_SP4 : BOOL; (* AT %MW10004.8 *) (* R361 1 M 차종9 SP4 *)
    R361_1_M_차종9_SP5 : BOOL; (* AT %MW10004.9 *) (* R361 1 M 차종9 SP5 *)
    R361_1_M_차종9_SP6 : BOOL; (* AT %MW10004.10 *) (* R361 1 M 차종9 SP6 *)
    R361_1_M_차종9_SP7 : BOOL; (* AT %MW10004.11 *) (* R361 1 M 차종9 SP7 *)
    R361_1_M_차종9_SP8 : BOOL; (* AT %MW10004.12 *) (* R361 1 M 차종9 SP8 *)
    R361_1_M_차종9_SP9 : BOOL; (* AT %MW10004.13 *) (* R361 1 M 차종9 SP9 *)
    R361_1_M_차종9_T_GDI : BOOL; (* AT %MW10004.4 *) (* R361 1 M 차종9 T GDI *)
    R361_1_M_차종_OPT1_R_RACK_무 : BOOL; (* AT %MW10005.3 *) (* R361 1 M 차종 OPT1 R RACK 무 *)
    R361_1_M_차종_OPT1_R_RACK_유 : BOOL; (* AT %MW10005.2 *) (* R361 1 M 차종 OPT1 R RACK 유 *)
    R361_1_M_차종_OPT1_S_REP_EATER_무 : BOOL; (* AT %MW10005.7 *) (* R361 1 M 차종 OPT1 S REP EATER 무 *)
    R361_1_M_차종_OPT1_S_REP_EATER_유 : BOOL; (* AT %MW10005.6 *) (* R361 1 M 차종 OPT1 S REP EATER 유 *)
    R361_1_M_차종_OPT1_VAN_무 : BOOL; (* AT %MW10005.9 *) (* R361 1 M 차종 OPT1 VAN 무 *)
    R361_1_M_차종_OPT1_VAN_유 : BOOL; (* AT %MW10005.8 *) (* R361 1 M 차종 OPT1 VAN 유 *)
    R361_1_M_차종_OPT1_슬라이딩_무 : BOOL; (* AT %MW10005.1 *) (* R361 1 M 차종 OPT1 슬라이딩 무 *)
    R361_1_M_차종_OPT1_슬라이딩_유 : BOOL; (* AT %MW10005.0 *) (* R361 1 M 차종 OPT1 슬라이딩 유 *)
    R361_1_M_차종_OPT1_폴딩_무 : BOOL; (* AT %MW10005.5 *) (* R361 1 M 차종 OPT1 폴딩 무 *)
    R361_1_M_차종_OPT1_폴딩_유 : BOOL; (* AT %MW10005.4 *) (* R361 1 M 차종 OPT1 폴딩 유 *)
    R361_1_M_차종_무 : BOOL; (* AT %MW1502.1 *)
    R361_1_M_차종_유 : BOOL; (* AT %MW1502.0 *)
    R361_2_M_SEQ : WORD; (* AT %MW10020 *) (* R361 2 M SEQ *)
    R361_2_M_차종1_AX : BOOL; (* AT %MW10021.0 *) (* R361 2 M 차종1 AX *)
    R361_2_M_차종1_B : BOOL; (* AT %MW10021.1 *) (* R361 2 M 차종1 B *)
    R361_2_M_차종1_C : BOOL; (* AT %MW10021.2 *) (* R361 2 M 차종1 C *)
    R361_2_M_차종1_D : BOOL; (* AT %MW10021.3 *) (* R361 2 M 차종1 D *)
    R361_2_M_차종1_E : BOOL; (* AT %MW10021.4 *) (* R361 2 M 차종1 E *)
    R361_2_M_차종1_F : BOOL; (* AT %MW10021.5 *) (* R361 2 M 차종1 F *)
    R361_2_M_차종1_G : BOOL; (* AT %MW10021.6 *) (* R361 2 M 차종1 G *)
    R361_2_M_차종1_H : BOOL; (* AT %MW10021.7 *) (* R361 2 M 차종1 H *)
    R361_2_M_차종2_3DR : BOOL; (* AT %MW10021.8 *) (* R361 2 M 차종2 3DR *)
    R361_2_M_차종2_4DR : BOOL; (* AT %MW10021.9 *) (* R361 2 M 차종2 4DR *)
    R361_2_M_차종2_5DR : BOOL; (* AT %MW10021.10 *) (* R361 2 M 차종2 5DR *)
    R361_2_M_차종2_SP1 : BOOL; (* AT %MW10021.12 *) (* R361 2 M 차종2 SP1 *)
    R361_2_M_차종2_SP2 : BOOL; (* AT %MW10021.13 *) (* R361 2 M 차종2 SP2 *)
    R361_2_M_차종2_WGN : BOOL; (* AT %MW10021.11 *) (* R361 2 M 차종2 WGN *)
    R361_2_M_차종3_LHD : BOOL; (* AT %MW10021.14 *) (* R361 2 M 차종3 LHD *)
    R361_2_M_차종3_RHD : BOOL; (* AT %MW10021.15 *) (* R361 2 M 차종3 RHD *)
    R361_2_M_차종4_EEC : BOOL; (* AT %MW10022.3 *) (* R361 2 M 차종4 EEC *)
    R361_2_M_차종4_SP1 : BOOL; (* AT %MW10022.8 *) (* R361 2 M 차종4 SP1 *)
    R361_2_M_차종4_SP2 : BOOL; (* AT %MW10022.9 *) (* R361 2 M 차종4 SP2 *)
    R361_2_M_차종4_SP3 : BOOL; (* AT %MW10022.11 *) (* R361 2 M 차종4 SP3 *)
    R361_2_M_차종4_SP4 : BOOL; (* AT %MW10022.12 *) (* R361 2 M 차종4 SP4 *)
    R361_2_M_차종4_SP5 : BOOL; (* AT %MW10022.13 *) (* R361 2 M 차종4 SP5 *)
    R361_2_M_차종4_SP6 : BOOL; (* AT %MW10022.14 *) (* R361 2 M 차종4 SP6 *)
    R361_2_M_차종4_SP7 : BOOL; (* AT %MW10022.15 *) (* R361 2 M 차종4 SP7 *)
    R361_2_M_차종4_내수 : BOOL; (* AT %MW10022.0 *) (* R361 2 M 차종4 내수 *)
    R361_2_M_차종4_러시아 : BOOL; (* AT %MW10022.10 *) (* R361 2 M 차종4 러시아 *)
    R361_2_M_차종4_북미 : BOOL; (* AT %MW10022.2 *) (* R361 2 M 차종4 북미 *)
    R361_2_M_차종4_브라질 : BOOL; (* AT %MW10022.7 *) (* R361 2 M 차종4 브라질 *)
    R361_2_M_차종4_수출 : BOOL; (* AT %MW10022.1 *) (* R361 2 M 차종4 수출 *)
    R361_2_M_차종4_중국 : BOOL; (* AT %MW10022.6 *) (* R361 2 M 차종4 중국 *)
    R361_2_M_차종4_중동 : BOOL; (* AT %MW10022.5 *) (* R361 2 M 차종4 중동 *)
    R361_2_M_차종4_호주 : BOOL; (* AT %MW10022.4 *) (* R361 2 M 차종4 호주 *)
    R361_2_M_차종5_AT : BOOL; (* AT %MW10023.1 *) (* R361 2 M 차종5 AT *)
    R361_2_M_차종5_MT : BOOL; (* AT %MW10023.0 *) (* R361 2 M 차종5 MT *)
    R361_2_M_차종5_SP1 : BOOL; (* AT %MW10023.2 *) (* R361 2 M 차종5 SP1 *)
    R361_2_M_차종6_DSROOF : BOOL; (* AT %MW10023.6 *) (* R361 2 M 차종6 DSROOF *)
    R361_2_M_차종6_SP1 : BOOL; (* AT %MW10023.7 *) (* R361 2 M 차종6 SP1 *)
    R361_2_M_차종6_썬루프 : BOOL; (* AT %MW10023.4 *) (* R361 2 M 차종6 썬루프 *)
    R361_2_M_차종6_일반루프 : BOOL; (* AT %MW10023.3 *) (* R361 2 M 차종6 일반루프 *)
    R361_2_M_차종6_파노라마루프 : BOOL; (* AT %MW10023.5 *) (* R361 2 M 차종6 파노라마루프 *)
    R361_2_M_차종7_DSL : BOOL; (* AT %MW10023.9 *) (* R361 2 M 차종7 DSL *)
    R361_2_M_차종7_GSL : BOOL; (* AT %MW10023.8 *) (* R361 2 M 차종7 GSL *)
    R361_2_M_차종7_SP1 : BOOL; (* AT %MW10023.10 *) (* R361 2 M 차종7 SP1 *)
    R361_2_M_차종7_SP2 : BOOL; (* AT %MW10023.11 *) (* R361 2 M 차종7 SP2 *)
    R361_2_M_차종7_SP3 : BOOL; (* AT %MW10023.12 *) (* R361 2 M 차종7 SP3 *)
    R361_2_M_차종7_SP4 : BOOL; (* AT %MW10023.13 *) (* R361 2 M 차종7 SP4 *)
    R361_2_M_차종7_SP5 : BOOL; (* AT %MW10023.14 *) (* R361 2 M 차종7 SP5 *)
    R361_2_M_차종7_SP6 : BOOL; (* AT %MW10023.15 *) (* R361 2 M 차종7 SP6 *)
    R361_2_M_차종8_2WD : BOOL; (* AT %MW10024.0 *) (* R361 2 M 차종8 2WD *)
    R361_2_M_차종8_4WD : BOOL; (* AT %MW10024.1 *) (* R361 2 M 차종8 4WD *)
    R361_2_M_차종8_SP1 : BOOL; (* AT %MW10024.2 *) (* R361 2 M 차종8 SP1 *)
    R361_2_M_차종9_MPI : BOOL; (* AT %MW10024.3 *) (* R361 2 M 차종9 MPI *)
    R361_2_M_차종9_SP1 : BOOL; (* AT %MW10024.5 *) (* R361 2 M 차종9 SP1 *)
    R361_2_M_차종9_SP10 : BOOL; (* AT %MW10024.14 *) (* R361 2 M 차종9 SP10 *)
    R361_2_M_차종9_SP11 : BOOL; (* AT %MW10024.15 *) (* R361 2 M 차종9 SP11 *)
    R361_2_M_차종9_SP2 : BOOL; (* AT %MW10024.6 *) (* R361 2 M 차종9 SP2 *)
    R361_2_M_차종9_SP3 : BOOL; (* AT %MW10024.7 *) (* R361 2 M 차종9 SP3 *)
    R361_2_M_차종9_SP4 : BOOL; (* AT %MW10024.8 *) (* R361 2 M 차종9 SP4 *)
    R361_2_M_차종9_SP5 : BOOL; (* AT %MW10024.9 *) (* R361 2 M 차종9 SP5 *)
    R361_2_M_차종9_SP6 : BOOL; (* AT %MW10024.10 *) (* R361 2 M 차종9 SP6 *)
    R361_2_M_차종9_SP7 : BOOL; (* AT %MW10024.11 *) (* R361 2 M 차종9 SP7 *)
    R361_2_M_차종9_SP8 : BOOL; (* AT %MW10024.12 *) (* R361 2 M 차종9 SP8 *)
    R361_2_M_차종9_SP9 : BOOL; (* AT %MW10024.13 *) (* R361 2 M 차종9 SP9 *)
    R361_2_M_차종9_T_GDI : BOOL; (* AT %MW10024.4 *) (* R361 2 M 차종9 T GDI *)
    R361_2_M_차종_OPT1_R_RACK_무 : BOOL; (* AT %MW10025.3 *) (* R361 2 M 차종 OPT1 R RACK 무 *)
    R361_2_M_차종_OPT1_R_RACK_유 : BOOL; (* AT %MW10025.2 *) (* R361 2 M 차종 OPT1 R RACK 유 *)
    R361_2_M_차종_OPT1_S_REP_EATER_무 : BOOL; (* AT %MW10025.7 *) (* R361 2 M 차종 OPT1 S REP EATER 무 *)
    R361_2_M_차종_OPT1_S_REP_EATER_유 : BOOL; (* AT %MW10025.6 *) (* R361 2 M 차종 OPT1 S REP EATER 유 *)
    R361_2_M_차종_OPT1_VAN_무 : BOOL; (* AT %MW10025.9 *) (* R361 2 M 차종 OPT1 VAN 무 *)
    R361_2_M_차종_OPT1_VAN_유 : BOOL; (* AT %MW10025.8 *) (* R361 2 M 차종 OPT1 VAN 유 *)
    R361_2_M_차종_OPT1_슬라이딩_무 : BOOL; (* AT %MW10025.1 *) (* R361 2 M 차종 OPT1 슬라이딩 무 *)
    R361_2_M_차종_OPT1_슬라이딩_유 : BOOL; (* AT %MW10025.0 *) (* R361 2 M 차종 OPT1 슬라이딩 유 *)
    R361_2_M_차종_OPT1_폴딩_무 : BOOL; (* AT %MW10025.5 *) (* R361 2 M 차종 OPT1 폴딩 무 *)
    R361_2_M_차종_OPT1_폴딩_유 : BOOL; (* AT %MW10025.4 *) (* R361 2 M 차종 OPT1 폴딩 유 *)
    R361_2_M_차종_무 : BOOL; (* AT %MW1502.3 *)
    R361_2_M_차종_유 : BOOL; (* AT %MW1502.2 *)
    ROOF_RACK_M_수동모드 : BOOL; (* AT %MW1500.3 *)
    ROOF_RACK_M_운전준비_ON : BOOL; (* AT %MW1500.0 *)
    ROOF_RACK_M_자동_START : BOOL; (* AT %MW1500.5 *)
    ROOF_RACK_M_자동_운전중 : BOOL; (* AT %MW1500.4 *)
    ROOF_RACK_M_자동모드 : BOOL; (* AT %MW1500.1 *)
    ROOF_RACK_M_작업완료_SET_PLS : BOOL; (* AT %MW1500.8 *)
    ROOF_RACK_M_작업완료_리셋_PLS : BOOL; (* AT %MW1500.9 *)
    ROOF_RACK_M_총괄_이상 : BOOL; (* AT %MW1509.0 *)
    S362_M_공정_차종_무 : BOOL; (* AT %MW1002.1 *) (* S362_M_공정_차종_무 *)
    S362_M_공정_차종_유 : BOOL; (* AT %MW1002.0 *) (* S362_M_공정_차종_유 *)
    S362_M_작업완료_SET_PLS : BOOL; (* AT %MW1000.8 *) (* S362 M 작업완료 SET PLS *)
    S362_M_작업완료_리셋_PLS : BOOL; (* AT %MW1000.9 *) (* S362 M 작업완료 리셋 PLS *)
    S364_M_수동모드 : BOOL; (* AT %MW2000.3 *) (* S364 선택 수동모드 *)
    S364_M_운전준비_ON : BOOL; (* AT %MW2000.0 *) (* S364 운전준비 ON *)
    S364_M_자동_START : BOOL; (* AT %MW2000.5 *) (* S364 자동운전중 *)
    S364_M_자동_운전중 : BOOL; (* AT %MW2000.4 *) (* S364 자동운전중 *)
    S364_M_자동모드 : BOOL; (* AT %MW2000.1 *) (* S364 선택 자동모드 *)
    S364_M_총괄_이상 : BOOL; (* AT %MW2009.0 *) (* S364_M_총괄_이상 *)
    전체_M_GATE_자동기동 : BOOL; (* AT %MW308.1 *) (* 전체_M_자동_운전 *)
    전체_라인_M_총괄_SAFETY_이상 : BOOL; (* AT %MW300.2 *) (* ALL공정 SAFETY  이상총괄 *)
    전체_라인_M_총괄_공기압_이상 : BOOL; (* AT %MW300.3 *) (* ALL공정 공기압 이상총괄 *)
    전체_라인_M_총괄_비상정지_이상 : BOOL; (* AT %MW300.1 *) (* ALL공정 비상정지 이상총괄 *)
END_VAR
VAR_EXTERNAL
    HOP_PBL_운전준비_ON : BOOL; (* AT %MW87500.0 *) (* HOP_PBL_운전준비_ON *)
    HOP_PLB_362_4_자동_운전 : BOOL; (* AT %MW87500.4 *) (* HOP PLB 362~4 자동기동 *)
    HOP_SSP_362_4_수동_선택 : BOOL; (* AT %MW87500.3 *) (* HOP 362~4 수동선택 *)
    HOP_SSP_362_4_자동_선택 : BOOL; (* AT %MW87500.2 *) (* HOP 362~4 자동선택 *)
    MCP_PBL_362_4_자동_운전 : BOOL; (* AT %MW87630.4 *) (* MCP PBL 362~4 자동기동 *)
    MCP_PBL_운전준비_ON : BOOL; (* AT %MW87630.0 *) (* MCP_PBL_운전준비_ON *)
    MCP_SPB_작업완료_RESET : BOOL; (* AT %MW87631.6 *) (* MCP_SPB_작업완료_RESET *)
    MCP_SPB_작업완료_SET : BOOL; (* AT %MW87631.7 *) (* MCP_SPB_작업완료_SET *)
    MCP_SSP_362_4_수동_선택 : BOOL; (* AT %MW87630.2 *) (* MCP 362~4 수동선택 *)
    MCP_SSP_362_4_자동_선택 : BOOL; (* AT %MW87630.3 *) (* MCP 362~4 자동동선택 *)
END_VAR
VAR
    ROOF_RACK_READY : TON;
    S364_READY : TON;
    T364_AUTO : TON;
    T_ROOF_RACK_AUTO : TON;
END_VAR
VAR
    _t1 : BOOL;
    _t2 : BOOL;
END_VAR

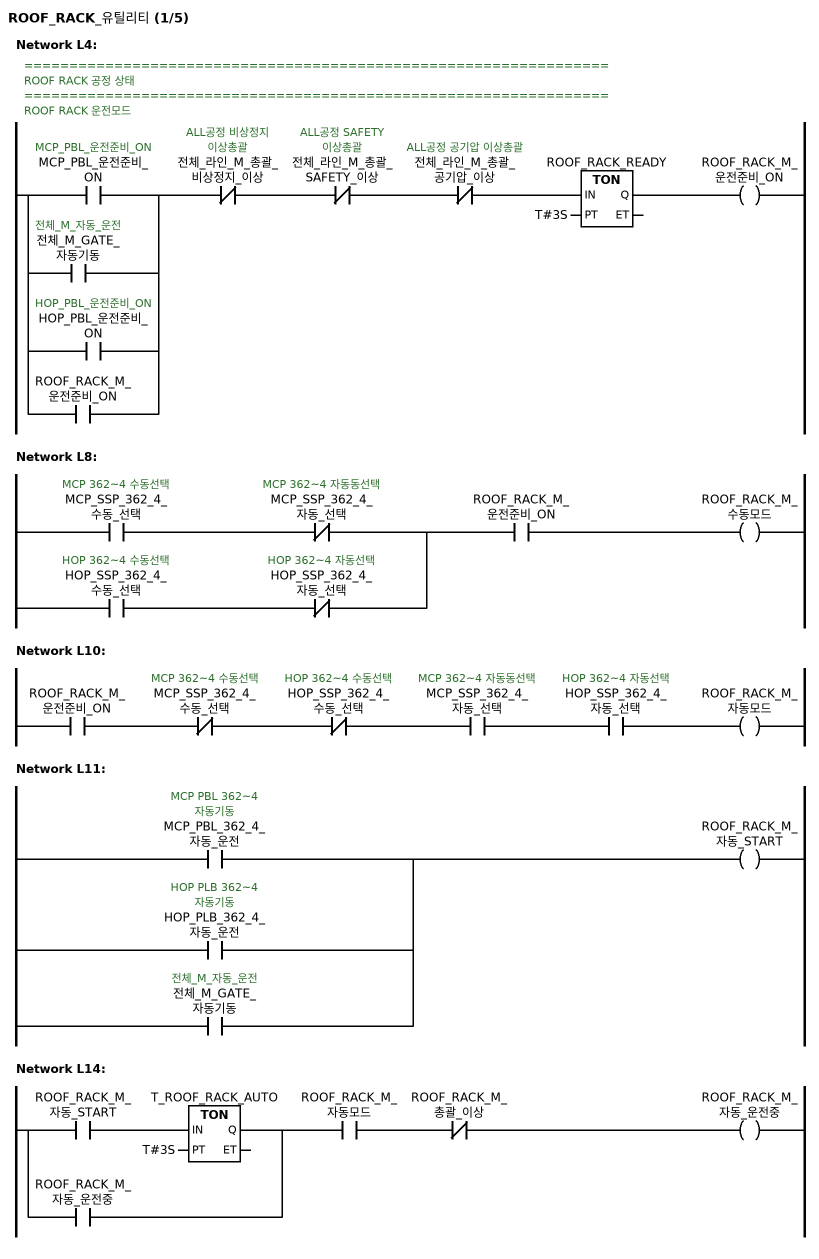
(* ================================================================= *)
(* ROOF RACK 공정 상태 *)
(* ================================================================= *)
(* ROOF RACK 운전모드 *)
(* Rung L4 *)
ROOF_RACK_READY(IN := (MCP_PBL_운전준비_ON OR 전체_M_GATE_자동기동 OR HOP_PBL_운전준비_ON OR ROOF_RACK_M_운전준비_ON) AND NOT 전체_라인_M_총괄_비상정지_이상 AND NOT 전체_라인_M_총괄_SAFETY_이상 AND NOT 전체_라인_M_총괄_공기압_이상, PT := T#3S);
ROOF_RACK_M_운전준비_ON := ROOF_RACK_READY.Q;
(* Rung L8 *)
ROOF_RACK_M_수동모드 := ((MCP_SSP_362_4_수동_선택 AND NOT MCP_SSP_362_4_자동_선택) OR (HOP_SSP_362_4_수동_선택 AND NOT HOP_SSP_362_4_자동_선택)) AND ROOF_RACK_M_운전준비_ON;
(* Rung L10 *)
ROOF_RACK_M_자동모드 := ROOF_RACK_M_운전준비_ON AND NOT MCP_SSP_362_4_수동_선택 AND NOT HOP_SSP_362_4_수동_선택 AND MCP_SSP_362_4_자동_선택 AND HOP_SSP_362_4_자동_선택;
(* Rung L11 *)
ROOF_RACK_M_자동_START := MCP_PBL_362_4_자동_운전 OR HOP_PLB_362_4_자동_운전 OR 전체_M_GATE_자동기동;
(* Rung L14 *)
T_ROOF_RACK_AUTO(IN := ROOF_RACK_M_자동_START, PT := T#3S);
ROOF_RACK_M_자동_운전중 := (T_ROOF_RACK_AUTO.Q OR ROOF_RACK_M_자동_운전중) AND ROOF_RACK_M_자동모드 AND NOT ROOF_RACK_M_총괄_이상;

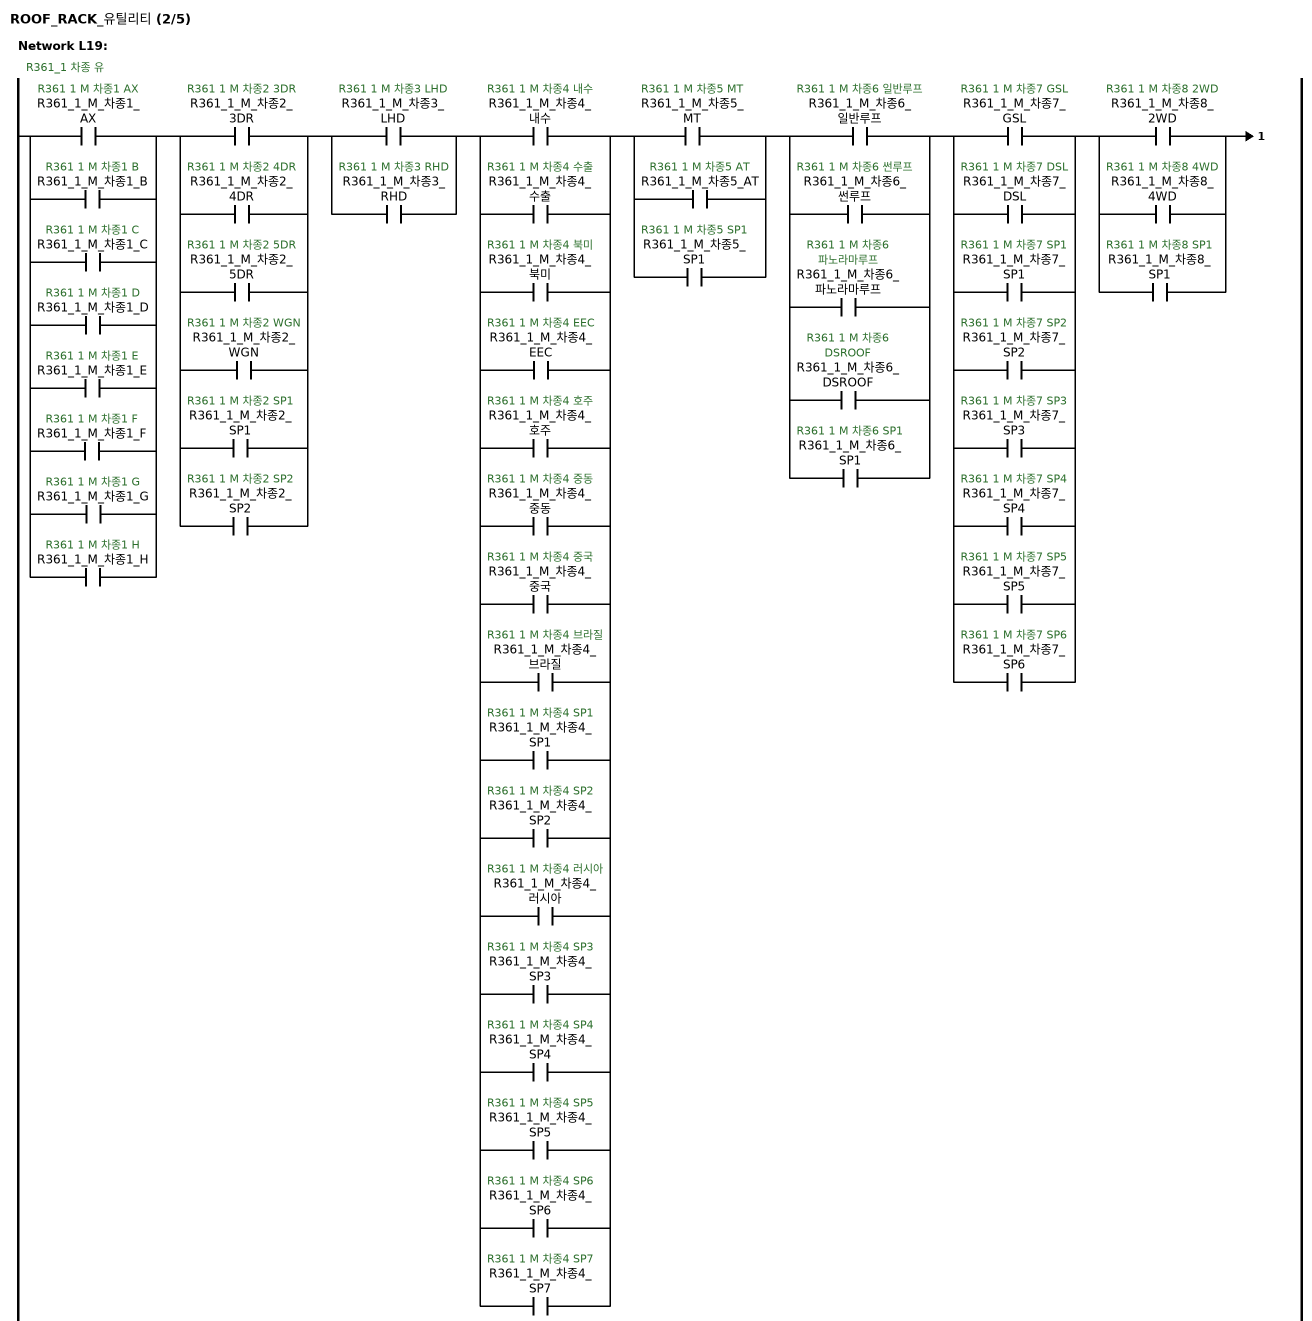

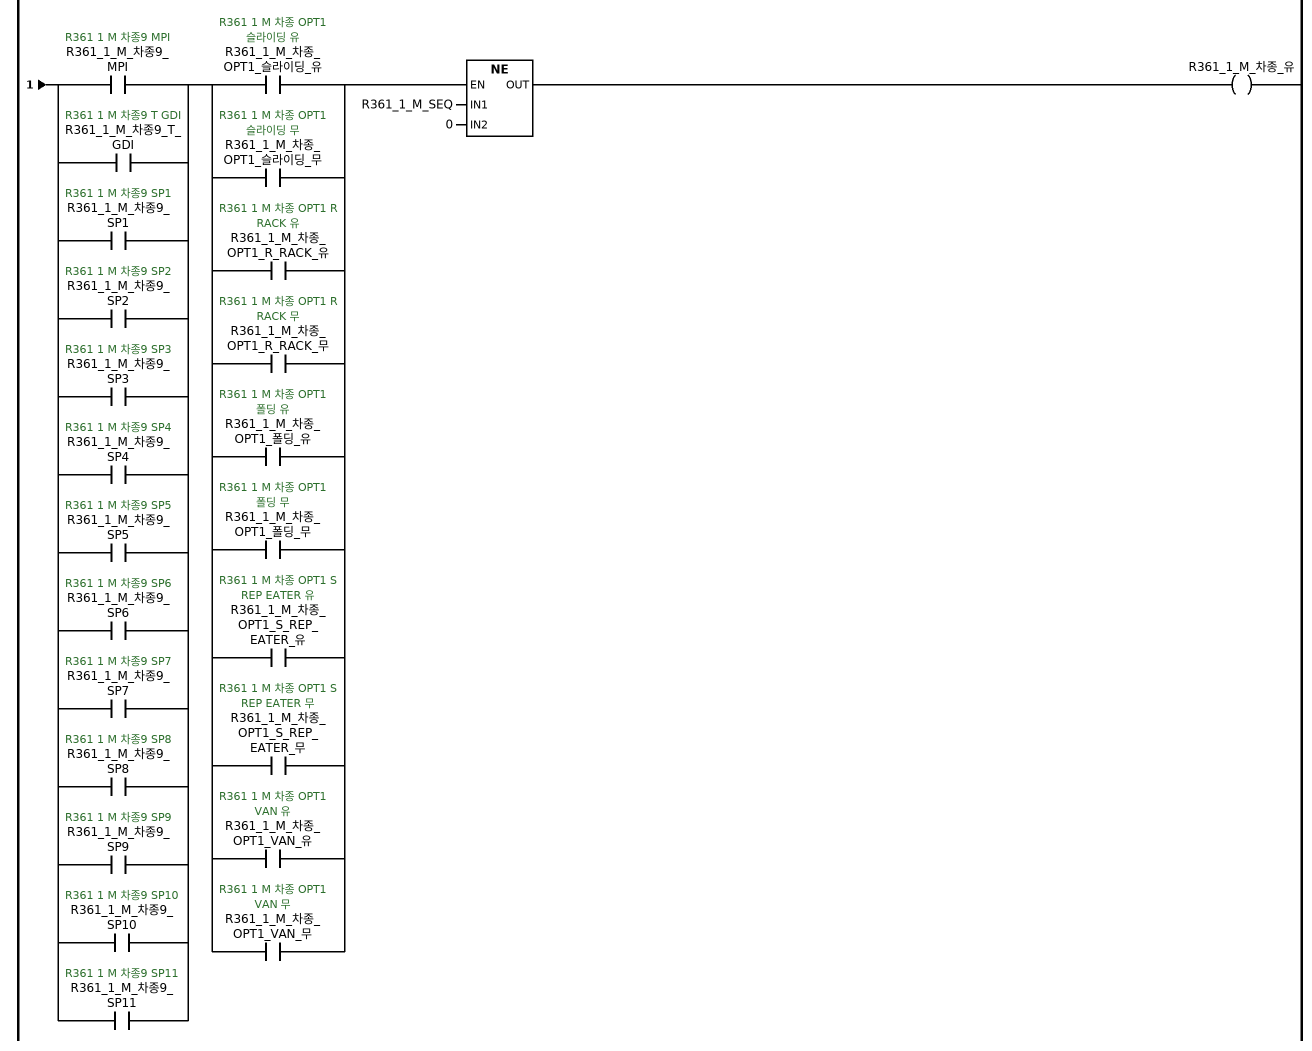
(* R361_1 차종 유 *)
(* Rung L19 *)
IF (R361_1_M_차종1_AX OR R361_1_M_차종1_B OR R361_1_M_차종1_C OR R361_1_M_차종1_D OR R361_1_M_차종1_E OR R361_1_M_차종1_F OR R361_1_M_차종1_G OR R361_1_M_차종1_H) AND (R361_1_M_차종2_3DR OR R361_1_M_차종2_4DR OR R361_1_M_차종2_5DR OR R361_1_M_차종2_WGN OR R361_1_M_차종2_SP1 OR R361_1_M_차종2_SP2) AND (R361_1_M_차종3_LHD OR R361_1_M_차종3_RHD) AND (R361_1_M_차종4_내수 OR R361_1_M_차종4_수출 OR R361_1_M_차종4_북미 OR R361_1_M_차종4_EEC OR R361_1_M_차종4_호주 OR R361_1_M_차종4_중동 OR R361_1_M_차종4_중국 OR R361_1_M_차종4_브라질 OR R361_1_M_차종4_SP1 OR R361_1_M_차종4_SP2 OR R361_1_M_차종4_러시아 OR R361_1_M_차종4_SP3 OR R361_1_M_차종4_SP4 OR R361_1_M_차종4_SP5 OR R361_1_M_차종4_SP6 OR R361_1_M_차종4_SP7) AND (R361_1_M_차종5_MT OR R361_1_M_차종5_AT OR R361_1_M_차종5_SP1) AND (R361_1_M_차종6_일반루프 OR R361_1_M_차종6_썬루프 OR R361_1_M_차종6_파노라마루프 OR R361_1_M_차종6_DSROOF OR R361_1_M_차종6_SP1) AND (R361_1_M_차종7_GSL OR R361_1_M_차종7_DSL OR R361_1_M_차종7_SP1 OR R361_1_M_차종7_SP2 OR R361_1_M_차종7_SP3 OR R361_1_M_차종7_SP4 OR R361_1_M_차종7_SP5 OR R361_1_M_차종7_SP6) AND (R361_1_M_차종8_2WD OR R361_1_M_차종8_4WD OR R361_1_M_차종8_SP1) AND (R361_1_M_차종9_MPI OR R361_1_M_차종9_T_GDI OR R361_1_M_차종9_SP1 OR R361_1_M_차종9_SP2 OR R361_1_M_차종9_SP3 OR R361_1_M_차종9_SP4 OR R361_1_M_차종9_SP5 OR R361_1_M_차종9_SP6 OR R361_1_M_차종9_SP7 OR R361_1_M_차종9_SP8 OR R361_1_M_차종9_SP9 OR R361_1_M_차종9_SP10 OR R361_1_M_차종9_SP11) AND (R361_1_M_차종_OPT1_슬라이딩_유 OR R361_1_M_차종_OPT1_슬라이딩_무 OR R361_1_M_차종_OPT1_R_RACK_유 OR R361_1_M_차종_OPT1_R_RACK_무 OR R361_1_M_차종_OPT1_폴딩_유 OR R361_1_M_차종_OPT1_폴딩_무 OR R361_1_M_차종_OPT1_S_REP_EATER_유 OR R361_1_M_차종_OPT1_S_REP_EATER_무 OR R361_1_M_차종_OPT1_VAN_유 OR R361_1_M_차종_OPT1_VAN_무) THEN
    _t1 := R361_1_M_SEQ <> 0;
END_IF;
R361_1_M_차종_유 := _t1;

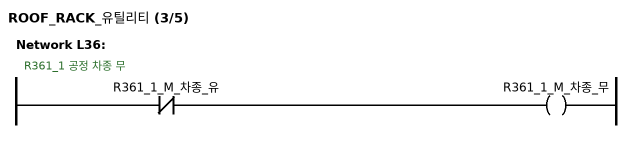
(* R361_1 공정 차종 무 *)
(* Rung L36 *)
R361_1_M_차종_무 := NOT R361_1_M_차종_유;

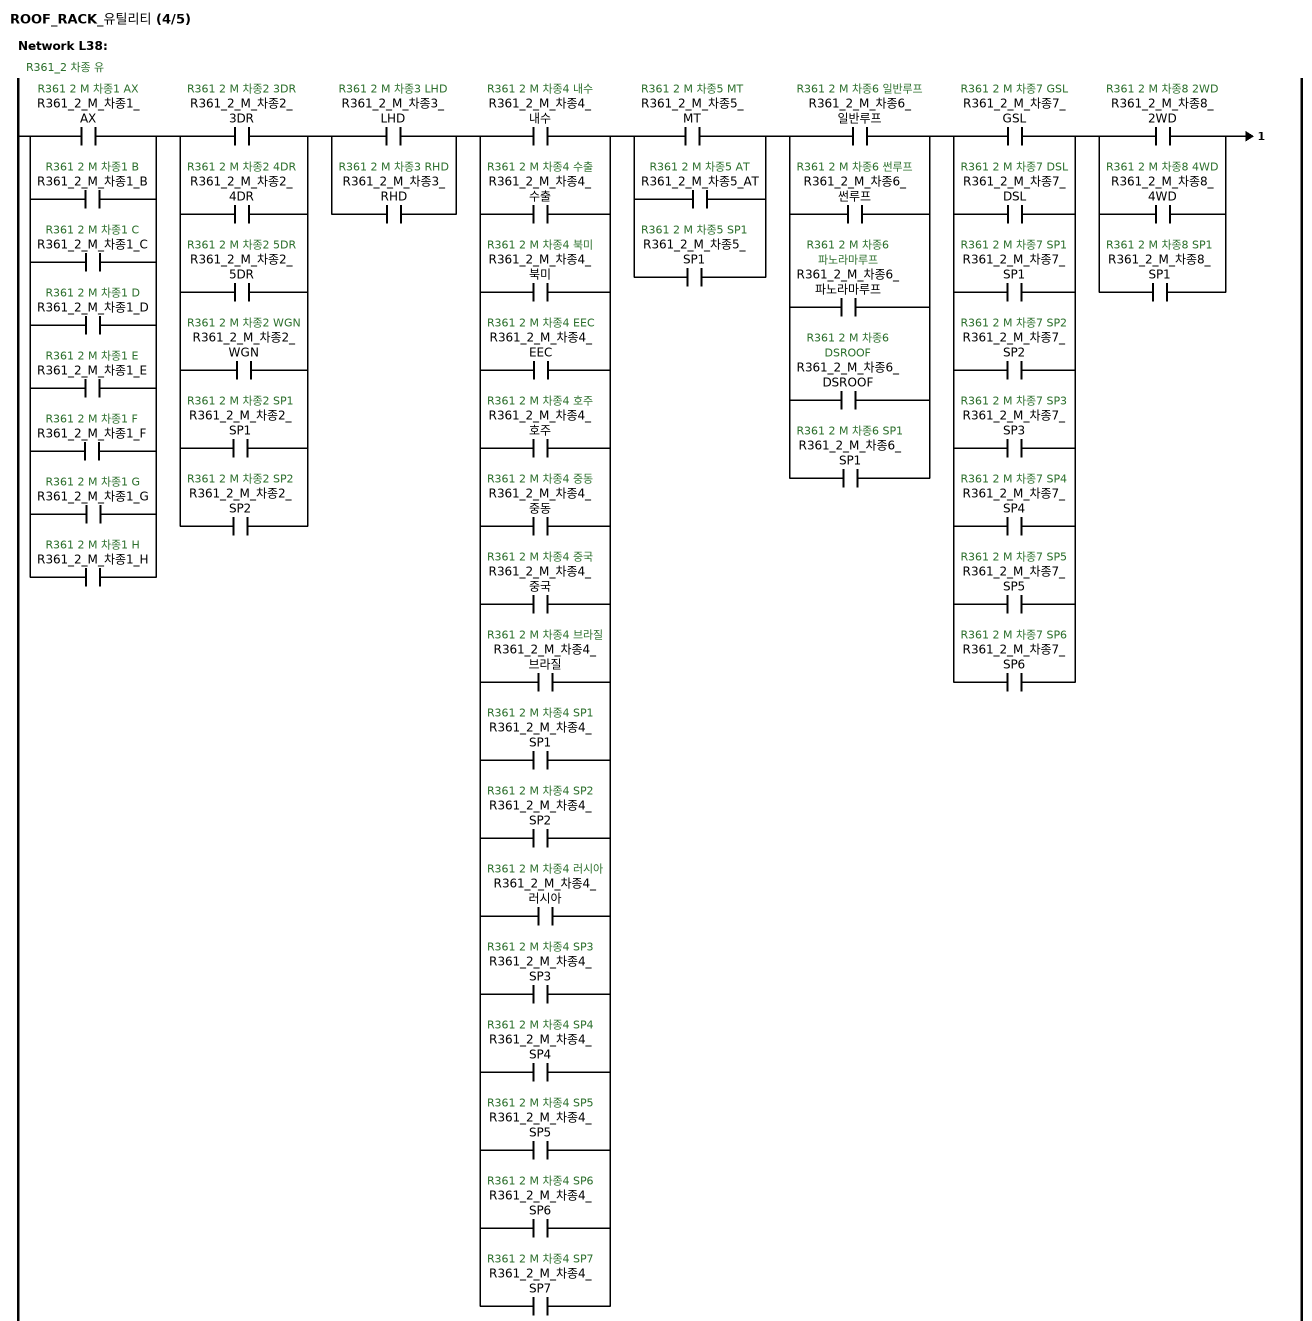

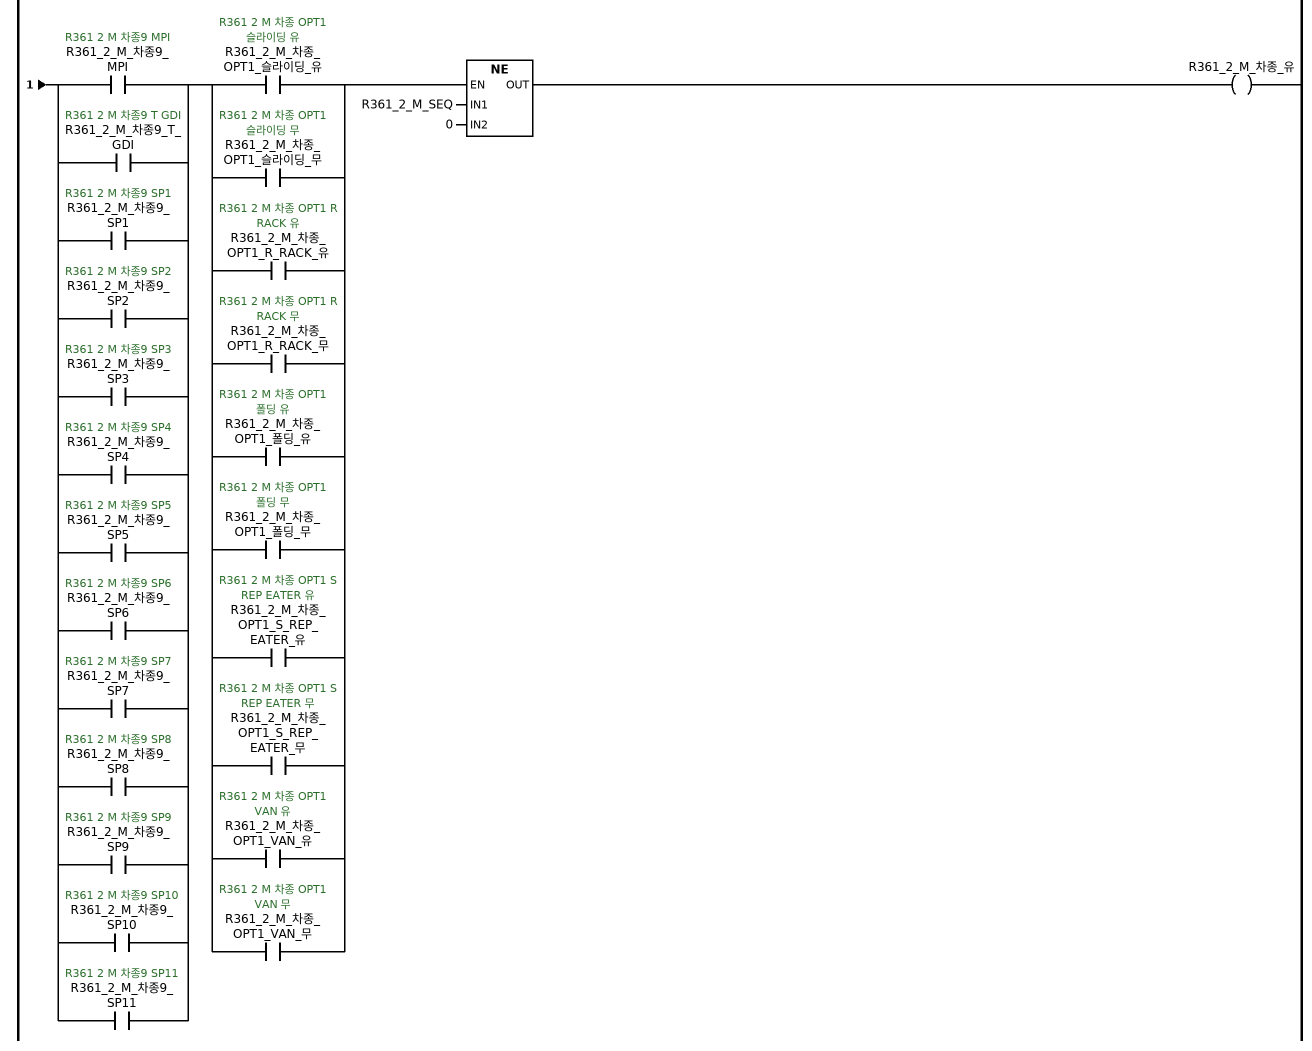
(* R361_2 차종 유 *)
(* Rung L38 *)
IF (R361_2_M_차종1_AX OR R361_2_M_차종1_B OR R361_2_M_차종1_C OR R361_2_M_차종1_D OR R361_2_M_차종1_E OR R361_2_M_차종1_F OR R361_2_M_차종1_G OR R361_2_M_차종1_H) AND (R361_2_M_차종2_3DR OR R361_2_M_차종2_4DR OR R361_2_M_차종2_5DR OR R361_2_M_차종2_WGN OR R361_2_M_차종2_SP1 OR R361_2_M_차종2_SP2) AND (R361_2_M_차종3_LHD OR R361_2_M_차종3_RHD) AND (R361_2_M_차종4_내수 OR R361_2_M_차종4_수출 OR R361_2_M_차종4_북미 OR R361_2_M_차종4_EEC OR R361_2_M_차종4_호주 OR R361_2_M_차종4_중동 OR R361_2_M_차종4_중국 OR R361_2_M_차종4_브라질 OR R361_2_M_차종4_SP1 OR R361_2_M_차종4_SP2 OR R361_2_M_차종4_러시아 OR R361_2_M_차종4_SP3 OR R361_2_M_차종4_SP4 OR R361_2_M_차종4_SP5 OR R361_2_M_차종4_SP6 OR R361_2_M_차종4_SP7) AND (R361_2_M_차종5_MT OR R361_2_M_차종5_AT OR R361_2_M_차종5_SP1) AND (R361_2_M_차종6_일반루프 OR R361_2_M_차종6_썬루프 OR R361_2_M_차종6_파노라마루프 OR R361_2_M_차종6_DSROOF OR R361_2_M_차종6_SP1) AND (R361_2_M_차종7_GSL OR R361_2_M_차종7_DSL OR R361_2_M_차종7_SP1 OR R361_2_M_차종7_SP2 OR R361_2_M_차종7_SP3 OR R361_2_M_차종7_SP4 OR R361_2_M_차종7_SP5 OR R361_2_M_차종7_SP6) AND (R361_2_M_차종8_2WD OR R361_2_M_차종8_4WD OR R361_2_M_차종8_SP1) AND (R361_2_M_차종9_MPI OR R361_2_M_차종9_T_GDI OR R361_2_M_차종9_SP1 OR R361_2_M_차종9_SP2 OR R361_2_M_차종9_SP3 OR R361_2_M_차종9_SP4 OR R361_2_M_차종9_SP5 OR R361_2_M_차종9_SP6 OR R361_2_M_차종9_SP7 OR R361_2_M_차종9_SP8 OR R361_2_M_차종9_SP9 OR R361_2_M_차종9_SP10 OR R361_2_M_차종9_SP11) AND (R361_2_M_차종_OPT1_슬라이딩_유 OR R361_2_M_차종_OPT1_슬라이딩_무 OR R361_2_M_차종_OPT1_R_RACK_유 OR R361_2_M_차종_OPT1_R_RACK_무 OR R361_2_M_차종_OPT1_폴딩_유 OR R361_2_M_차종_OPT1_폴딩_무 OR R361_2_M_차종_OPT1_S_REP_EATER_유 OR R361_2_M_차종_OPT1_S_REP_EATER_무 OR R361_2_M_차종_OPT1_VAN_유 OR R361_2_M_차종_OPT1_VAN_무) THEN
    _t2 := R361_2_M_SEQ <> 0;
END_IF;
R361_2_M_차종_유 := _t2;

